LIN {X 0,Y 573.685,Z 492.708,A -85,B 0,C 180,E1 -2287.223,E2 -2287.223} C_VEL
LIN {X 0,Y 573.847,Z 485.027,A -85,B 0,C 180,E1 -2290.013,E2 -2290.013} C_VEL
LIN {X 0,Y 573.778,Z 480.732,A -85,B 0,C 180,E1 -2291.655,E2 -2291.655} C_VEL
LIN {X 0,Y 573.25,Z 477.707,A -85,B 0,C 180,E1 -2292.971,E2 -2292.971} C_VEL
LIN {X 0,Y 573.232,Z 477.709,A -85,B 0,C 180,E1 -2295.666,E2 -2295.666} C_VEL
LIN {X 0,Y 573.254,Z 477.706,A -85,B 0,C 180,E1 -2298.545,E2 -2298.545} C_VEL
LIN {X 0,Y 573.245,Z 477.706,A -85,B 0,C 180,E1 -2301.299,E2 -2301.299} C_VEL
LIN {X 0,Y 573.257,Z 477.705,A -85,B 0,C 180,E1 -2304.01,E2 -2304.01} C_VEL
LIN {X 0,Y 573.275,Z 477.704,A -85,B 0,C 180,E1 -2306.518,E2 -2306.518} C_VEL
LIN {X 0,Y 573.237,Z 477.707,A -85,B 0,C 180,E1 -2309.114,E2 -2309.114} C_VEL
LIN {X 0,Y 573.256,Z 477.706,A -85,B 0,C 180,E1 -2311.968,E2 -2311.968} C_VEL
LIN {X 0,Y 573.25,Z 477.705,A -85,B 0,C 180,E1 -2314.59,E2 -2314.59} C_VEL
LIN {X 0,Y 573.23,Z 477.709,A -85,B 0,C 180,E1 -2317.662,E2 -2317.662} C_VEL
LIN {X 0,Y 573.25,Z 477.706,A -85,B 0,C 180,E1 -2319.924,E2 -2319.924} C_VEL
LIN {X 0,Y 573.254,Z 477.707,A -85,B 0,C 180,E1 -2322.988,E2 -2322.988} C_VEL
LIN {X 0,Y 573.263,Z 477.704,A -85,B 0,C 180,E1 -2325.807,E2 -2325.807} C_VEL
LIN {X 0,Y 573.272,Z 477.703,A -85,B 0,C 180,E1 -2328.734,E2 -2328.734} C_VEL
LIN {X 0,Y 573.301,Z 477.7,A -85,B 0,C 180,E1 -2331.541,E2 -2331.541} C_VEL
LIN {X 0,Y 573.288,Z 477.7,A -85,B 0,C 180,E1 -2334.372,E2 -2334.372} C_VEL
LIN {X 0,Y 573.302,Z 477.699,A -85,B 0,C 180,E1 -2337.893,E2 -2337.893} C_VEL
LIN {X 0,Y 573.33,Z 477.697,A -85,B 0,C 180,E1 -2340.703,E2 -2340.703} C_VEL
LIN {X 0,Y 573.239,Z 477.707,A -85,B 0,C 180,E1 -2343.515,E2 -2343.515} C_VEL
LIN {X 0,Y 573.298,Z 477.699,A -85,B 0,C 180,E1 -2345.628,E2 -2345.628} C_VEL
LIN {X 0,Y 573.3,Z 477.7,A -85,B 0,C 180,E1 -2348.46,E2 -2348.46} C_VEL
LIN {X 0,Y 573.289,Z 477.701,A -85,B 0,C 180,E1 -2351.312,E2 -2351.312} C_VEL
LIN {X 0,Y 573.272,Z 477.702,A -85,B 0,C 180,E1 -2354.425,E2 -2354.425} C_VEL
LIN {X 0,Y 573.252,Z 477.707,A -85,B 0,C 180,E1 -2357.112,E2 -2357.112} C_VEL
LIN {X 0,Y 573.25,Z 477.706,A -85,B 0,C 180,E1 -2360.077,E2 -2360.077} C_VEL
LIN {X 0,Y 573.231,Z 477.708,A -85,B 0,C 180,E1 -2362.338,E2 -2362.338} C_VEL
LIN {X 0,Y 573.244,Z 477.706,A -85,B 0,C 180,E1 -2364.402,E2 -2364.402} C_VEL
LIN {X 0,Y 572.619,Z 477.786,A -85,B 0,C 180,E1 -2364.989,E2 -2364.989} C_VEL
LIN {X 0,Y 569.783,Z 478.14,A -85,B 0,C 180,E1 -2365.941,E2 -2365.941} C_VEL
LIN {X 0,Y 567.356,Z 478.442,A -85,B 0,C 180,E1 -2366.707,E2 -2366.707} C_VEL
LIN {X 0,Y 566.303,Z 478.572,A -85,B 0,C 180,E1 -2367.298,E2 -2367.298} C_VEL
LIN {X 0,Y 566.213,Z 478.581,A -85,B 0,C 180,E1 -2367.498,E2 -2367.498} C_VEL
LIN {X 0,Y 566.188,Z 478.585,A -85,B 0,C 180,E1 -2370.593,E2 -2370.593} C_VEL
LIN {X 0,Y 566.223,Z 478.58,A -85,B 0,C 180,E1 -2373.102,E2 -2373.102} C_VEL
LIN {X 0,Y 566.208,Z 478.584,A -85,B 0,C 180,E1 -2375.689,E2 -2375.689} C_VEL
LIN {X 0,Y 566.213,Z 478.581,A -85,B 0,C 180,E1 -2378.56,E2 -2378.56} C_VEL
LIN {X 0,Y 566.217,Z 478.582,A -85,B 0,C 180,E1 -2381.136,E2 -2381.136} C_VEL
LIN {X 0,Y 566.197,Z 478.584,A -85,B 0,C 180,E1 -2384.036,E2 -2384.036} C_VEL
LIN {X 0,Y 566.203,Z 478.584,A -85,B 0,C 180,E1 -2387.083,E2 -2387.083} C_VEL
LIN {X 0,Y 566.226,Z 478.581,A -85,B 0,C 180,E1 -2389.804,E2 -2389.804} C_VEL
LIN {X 0,Y 566.199,Z 478.584,A -85,B 0,C 180,E1 -2392.6,E2 -2392.6} C_VEL
LIN {X 0,Y 566.21,Z 478.582,A -85,B 0,C 180,E1 -2395.183,E2 -2395.183} C_VEL
LIN {X 0,Y 566.234,Z 478.581,A -85,B 0,C 180,E1 -2397.745,E2 -2397.745} C_VEL
LIN {X 0,Y 566.205,Z 478.582,A -85,B 0,C 180,E1 -2400.329,E2 -2400.329} C_VEL
LIN {X 0,Y 566.227,Z 478.579,A -85,B 0,C 180,E1 -2402.663,E2 -2402.663} C_VEL
LIN {X 0,Y 566.239,Z 478.578,A -85,B 0,C 180,E1 -2405.04,E2 -2405.04} C_VEL
LIN {X 0,Y 566.197,Z 478.583,A -85,B 0,C 180,E1 -2408.138,E2 -2408.138} C_VEL
LIN {X 0,Y 566.234,Z 478.578,A -85,B 0,C 180,E1 -2410.615,E2 -2410.615} C_VEL
LIN {X 0,Y 566.221,Z 478.582,A -85,B 0,C 180,E1 -2413.413,E2 -2413.413} C_VEL
LIN {X 0,Y 566.202,Z 478.584,A -85,B 0,C 180,E1 -2416.36,E2 -2416.36} C_VEL
LIN {X 0,Y 566.24,Z 478.58,A -85,B 0,C 180,E1 -2418.676,E2 -2418.676} C_VEL
LIN {X 0,Y 566.21,Z 478.582,A -85,B 0,C 180,E1 -2421.435,E2 -2421.435} C_VEL
LIN {X 0,Y 566.263,Z 478.577,A -85,B 0,C 180,E1 -2424.302,E2 -2424.302} C_VEL
LIN {X 0,Y 566.287,Z 478.573,A -85,B 0,C 180,E1 -2427.867,E2 -2427.867} C_VEL
LIN {X 0,Y 566.307,Z 478.571,A -85,B 0,C 180,E1 -2430.711,E2 -2430.711} C_VEL
LIN {X 0,Y 566.07,Z 478.602,A -85,B 0,C 180,E1 -2432.847,E2 -2432.847} C_VEL
LIN {X 0,Y 566.013,Z 478.622,A -85,B 0,C 180,E1 -2433.56,E2 -2433.56} C_VEL
LIN {X 0,Y 566.008,Z 480.702,A -85,B 0,C 180,E1 -2435.701,E2 -2435.701} C_VEL
LIN {X 0,Y 566.007,Z 483.486,A -85,B 0,C 180,E1 -2438.569,E2 -2438.569} C_VEL
LIN {X 0,Y 565.951,Z 486.311,A -85,B 0,C 180,E1 -2441.46,E2 -2441.46} C_VEL
LIN {X 0,Y 565.962,Z 489.393,A -85,B 0,C 180,E1 -2444.397,E2 -2444.397} C_VEL
LIN {X 0,Y 565.88,Z 492.716,A -85,B 0,C 180,E1 -2447.342,E2 -2447.342} C_VEL
LIN {X 0,Y 565.863,Z 496.182,A -85,B 0,C 180,E1 -2450.35,E2 -2450.35} C_VEL
LIN {X 0,Y 565.875,Z 498.386,A -85,B 0,C 180,E1 -2452.235,E2 -2452.235} C_VEL
LIN {X 0,Y 567.913,Z 507.747,A -85,B 0,C 180,E1 -2452.463,E2 -2452.463} C_VEL
LIN {X 0,Y 567.775,Z 523.279,A -85,B 0,C 180,E1 -2452.841,E2 -2452.841} C_VEL
LIN {X 0,Y 567.567,Z 537.926,A -85,B 0,C 180,E1 -2453.344,E2 -2453.344} C_VEL
LIN {X 0,Y 567.393,Z 551.473,A -85,B 0,C 180,E1 -2453.948,E2 -2453.948} C_VEL
LIN {X 0,Y 567.1,Z 565.407,A -85,B 0,C 180,E1 -2454.725,E2 -2454.725} C_VEL
LIN {X 0,Y 566.884,Z 578.74,A -85,B 0,C 180,E1 -2455.64,E2 -2455.64} C_VEL
LIN {X 0,Y 566.645,Z 591.048,A -85,B 0,C 180,E1 -2456.66,E2 -2456.66} C_VEL
LIN {X 0,Y 566.423,Z 601.892,A -85,B 0,C 180,E1 -2457.729,E2 -2457.729} C_VEL
LIN {X 0,Y 566.247,Z 612.279,A -85,B 0,C 180,E1 -2458.95,E2 -2458.95} C_VEL
LIN {X 0,Y 566.152,Z 621.068,A -85,B 0,C 180,E1 -2460.182,E2 -2460.182} C_VEL
LIN {X 0,Y 566.038,Z 629.621,A -85,B 0,C 180,E1 -2461.64,E2 -2461.64} C_VEL
LIN {X 0,Y 565.941,Z 636.591,A -85,B 0,C 180,E1 -2463.12,E2 -2463.12} C_VEL
LIN {X 0,Y 565.905,Z 641.383,A -85,B 0,C 180,E1 -2464.407,E2 -2464.407} C_VEL
LIN {X 0,Y 565.841,Z 645.15,A -85,B 0,C 180,E1 -2465.715,E2 -2465.715} C_VEL
LIN {X 0,Y 565.854,Z 647.11,A -85,B 0,C 180,E1 -2466.596,E2 -2466.596} C_VEL
LIN {X 0,Y 565.832,Z 648.638,A -85,B 0,C 180,E1 -2467.489,E2 -2467.489} C_VEL
LIN {X 0,Y 565.816,Z 649.833,A -85,B 0,C 180,E1 -2468.507,E2 -2468.507} C_VEL
LIN {X 0,Y 565.847,Z 650.418,A -85,B 0,C 180,E1 -2469.64,E2 -2469.64} C_VEL
LIN {X 0,Y 565.856,Z 650.112,A -85,B 0,C 180,E1 -2471.167,E2 -2471.167} C_VEL
LIN {X 0,Y 565.865,Z 649.261,A -85,B 0,C 180,E1 -2472.119,E2 -2472.119} C_VEL
LIN {X 0,Y 565.854,Z 647.882,A -85,B 0,C 180,E1 -2473.087,E2 -2473.087} C_VEL
LIN {X 0,Y 565.895,Z 644.84,A -85,B 0,C 180,E1 -2474.499,E2 -2474.499} C_VEL
LIN {X 0,Y 565.906,Z 640.511,A -85,B 0,C 180,E1 -2475.935,E2 -2475.935} C_VEL
LIN {X 0,Y 565.984,Z 636.025,A -85,B 0,C 180,E1 -2477.106,E2 -2477.106} C_VEL
LIN {X 0,Y 566.025,Z 629.345,A -85,B 0,C 180,E1 -2478.505,E2 -2478.505} C_VEL
LIN {X 0,Y 566.122,Z 621.792,A -85,B 0,C 180,E1 -2479.793,E2 -2479.793} C_VEL
LIN {X 0,Y 566.251,Z 612.523,A -85,B 0,C 180,E1 -2481.107,E2 -2481.107} C_VEL
LIN {X 0,Y 566.436,Z 602.143,A -85,B 0,C 180,E1 -2482.333,E2 -2482.333} C_VEL
LIN {X 0,Y 566.674,Z 590.668,A -85,B 0,C 180,E1 -2483.465,E2 -2483.465} C_VEL
LIN {X 0,Y 566.897,Z 578.806,A -85,B 0,C 180,E1 -2484.444,E2 -2484.444} C_VEL
LIN {X 0,Y 567.089,Z 567.299,A -85,B 0,C 180,E1 -2485.243,E2 -2485.243} C_VEL
LIN {X 0,Y 567.331,Z 553.585,A -85,B 0,C 180,E1 -2486.033,E2 -2486.033} C_VEL
LIN {X 0,Y 567.545,Z 539.884,A -85,B 0,C 180,E1 -2486.667,E2 -2486.667} C_VEL
LIN {X 0,Y 567.769,Z 524.257,A -85,B 0,C 180,E1 -2487.219,E2 -2487.219} C_VEL
LIN {X 0,Y 567.921,Z 508.637,A -85,B 0,C 180,E1 -2487.609,E2 -2487.609} C_VEL
LIN {X 0,Y 567.681,Z 506.099,A -85,B 0,C 180,E1 -2487.668,E2 -2487.668} C_VEL
LIN {X 0,Y 565.879,Z 498.374,A -85,B 0,C 180,E1 -2487.865,E2 -2487.865} C_VEL
LIN {X 0,Y 565.878,Z 495.432,A -85,B 0,C 180,E1 -2490.385,E2 -2490.385} C_VEL
LIN {X 0,Y 565.901,Z 491.926,A -85,B 0,C 180,E1 -2493.443,E2 -2493.443} C_VEL
LIN {X 0,Y 565.903,Z 489.271,A -85,B 0,C 180,E1 -2495.805,E2 -2495.805} C_VEL
LIN {X 0,Y 565.901,Z 486.833,A -85,B 0,C 180,E1 -2498.125,E2 -2498.125} C_VEL
LIN {X 0,Y 566.007,Z 484.648,A -85,B 0,C 180,E1 -2500.677,E2 -2500.677} C_VEL
LIN {X 0,Y 566.067,Z 482.103,A -85,B 0,C 180,E1 -2503.408,E2 -2503.408} C_VEL
LIN {X 0,Y 566.052,Z 479.234,A -85,B 0,C 180,E1 -2506.355,E2 -2506.355} C_VEL
LIN {X 0,Y 566.061,Z 478.604,A -85,B 0,C 180,E1 -2507.086,E2 -2507.086} C_VEL
LIN {X 0,Y 566.238,Z 478.574,A -85,B 0,C 180,E1 -2509.27,E2 -2509.27} C_VEL
LIN {X 0,Y 566.236,Z 478.58,A -85,B 0,C 180,E1 -2512.153,E2 -2512.153} C_VEL
LIN {X 0,Y 566.283,Z 478.567,A -85,B 0,C 180,E1 -2515.016,E2 -2515.016} C_VEL
LIN {X 0,Y 566.279,Z 478.574,A -85,B 0,C 180,E1 -2517.866,E2 -2517.866} C_VEL
LIN {X 0,Y 566.301,Z 478.565,A -85,B 0,C 180,E1 -2520.711,E2 -2520.711} C_VEL
LIN {X 0,Y 566.273,Z 478.57,A -85,B 0,C 180,E1 -2522.845,E2 -2522.845} C_VEL
LIN {X 0,Y 566.258,Z 478.573,A -85,B 0,C 180,E1 -2525.698,E2 -2525.698} C_VEL
LIN {X 0,Y 566.231,Z 478.575,A -85,B 0,C 180,E1 -2528.565,E2 -2528.565} C_VEL
LIN {X 0,Y 566.247,Z 478.574,A -85,B 0,C 180,E1 -2531.454,E2 -2531.454} C_VEL
LIN {X 0,Y 566.229,Z 478.578,A -85,B 0,C 180,E1 -2534.506,E2 -2534.506} C_VEL
LIN {X 0,Y 566.195,Z 478.579,A -85,B 0,C 180,E1 -2537.332,E2 -2537.332} C_VEL
LIN {X 0,Y 566.215,Z 478.581,A -85,B 0,C 180,E1 -2540.337,E2 -2540.337} C_VEL
LIN {X 0,Y 566.185,Z 478.579,A -85,B 0,C 180,E1 -2543.404,E2 -2543.404} C_VEL
LIN {X 0,Y 566.222,Z 478.577,A -85,B 0,C 180,E1 -2545.748,E2 -2545.748} C_VEL
LIN {X 0,Y 566.204,Z 478.585,A -85,B 0,C 180,E1 -2548.203,E2 -2548.203} C_VEL
LIN {X 0,Y 566.19,Z 478.58,A -85,B 0,C 180,E1 -2550.592,E2 -2550.592} C_VEL
LIN {X 0,Y 566.226,Z 478.575,A -85,B 0,C 180,E1 -2553.102,E2 -2553.102} C_VEL
LIN {X 0,Y 566.21,Z 478.585,A -85,B 0,C 180,E1 -2555.688,E2 -2555.688} C_VEL
LIN {X 0,Y 566.213,Z 478.575,A -85,B 0,C 180,E1 -2558.559,E2 -2558.559} C_VEL
LIN {X 0,Y 566.209,Z 478.581,A -85,B 0,C 180,E1 -2561.136,E2 -2561.136} C_VEL
LIN {X 0,Y 566.198,Z 478.581,A -85,B 0,C 180,E1 -2564.036,E2 -2564.036} C_VEL
LIN {X 0,Y 566.219,Z 478.637,A -85,B 0,C 180,E1 -2566.948,E2 -2566.948} C_VEL
LIN {X 0,Y 566.854,Z 483.368,A -85,B 0,C 180,E1 -2568.921,E2 -2568.921} C_VEL
LIN {X 0,Y 566.738,Z 489.853,A -85,B 0,C 180,E1 -2571.375,E2 -2571.375} C_VEL
LIN {X 0,Y 566.643,Z 498.211,A -85,B 0,C 180,E1 -2574.343,E2 -2574.343} C_VEL
LIN {X 0,Y 566.532,Z 505.812,A -85,B 0,C 180,E1 -2576.919,E2 -2576.919} C_VEL
LIN {X 0,Y 566.54,Z 513.738,A -85,B 0,C 180,E1 -2579.429,E2 -2579.429} C_VEL
LIN {X 0,Y 566.491,Z 521.49,A -85,B 0,C 180,E1 -2581.873,E2 -2581.873} C_VEL
LIN {X 0,Y 566.363,Z 530.126,A -85,B 0,C 180,E1 -2584.644,E2 -2584.644} C_VEL
LIN {X 0,Y 566.244,Z 538.819,A -85,B 0,C 180,E1 -2587.371,E2 -2587.371} C_VEL
LIN {X 0,Y 566.185,Z 547.483,A -85,B 0,C 180,E1 -2590.041,E2 -2590.041} C_VEL
LIN {X 0,Y 566.124,Z 554.42,A -85,B 0,C 180,E1 -2592.145,E2 -2592.145} C_VEL
LIN {X 0,Y 568.001,Z 563.349,A -85,B 0,C 180,E1 -2592.339,E2 -2592.339} C_VEL
LIN {X 0,Y 567.825,Z 577.885,A -85,B 0,C 180,E1 -2592.647,E2 -2592.647} C_VEL
LIN {X 0,Y 567.7,Z 592.206,A -85,B 0,C 180,E1 -2593.087,E2 -2593.087} C_VEL
LIN {X 0,Y 567.499,Z 605.82,A -85,B 0,C 180,E1 -2593.636,E2 -2593.636} C_VEL
LIN {X 0,Y 567.213,Z 620.1,A -85,B 0,C 180,E1 -2594.366,E2 -2594.366} C_VEL
LIN {X 0,Y 566.973,Z 633.394,A -85,B 0,C 180,E1 -2595.208,E2 -2595.208} C_VEL
LIN {X 0,Y 566.757,Z 646.161,A -85,B 0,C 180,E1 -2596.19,E2 -2596.19} C_VEL
LIN {X 0,Y 566.545,Z 657.97,A -85,B 0,C 180,E1 -2597.28,E2 -2597.28} C_VEL
LIN {X 0,Y 566.343,Z 667.9,A -85,B 0,C 180,E1 -2598.366,E2 -2598.366} C_VEL
LIN {X 0,Y 566.204,Z 677.618,A -85,B 0,C 180,E1 -2599.631,E2 -2599.631} C_VEL
LIN {X 0,Y 566.08,Z 685.72,A -85,B 0,C 180,E1 -2600.892,E2 -2600.892} C_VEL
LIN {X 0,Y 566.014,Z 692.424,A -85,B 0,C 180,E1 -2602.15,E2 -2602.15} C_VEL
LIN {X 0,Y 565.943,Z 698.606,A -85,B 0,C 180,E1 -2603.583,E2 -2603.583} C_VEL
LIN {X 0,Y 565.866,Z 703.384,A -85,B 0,C 180,E1 -2605.012,E2 -2605.012} C_VEL
LIN {X 0,Y 565.909,Z 706.888,A -85,B 0,C 180,E1 -2606.44,E2 -2606.44} C_VEL
LIN {X 0,Y 565.836,Z 709.192,A -85,B 0,C 180,E1 -2607.864,E2 -2607.864} C_VEL
LIN {X 0,Y 565.838,Z 710.349,A -85,B 0,C 180,E1 -2609.288,E2 -2609.288} C_VEL
LIN {X 0,Y 565.838,Z 710.349,A -85,B 0,C 180,E1 -2610.711,E2 -2610.711} C_VEL
LIN {X 0,Y 565.836,Z 709.191,A -85,B 0,C 180,E1 -2612.135,E2 -2612.135} C_VEL
LIN {X 0,Y 565.909,Z 706.888,A -85,B 0,C 180,E1 -2613.56,E2 -2613.56} C_VEL
LIN {X 0,Y 565.866,Z 703.386,A -85,B 0,C 180,E1 -2614.987,E2 -2614.987} C_VEL
LIN {X 0,Y 565.956,Z 699.926,A -85,B 0,C 180,E1 -2616.059,E2 -2616.059} C_VEL
LIN {X 0,Y 565.999,Z 694.09,A -85,B 0,C 180,E1 -2617.491,E2 -2617.491} C_VEL
LIN {X 0,Y 566.057,Z 686.733,A -85,B 0,C 180,E1 -2618.928,E2 -2618.928} C_VEL
LIN {X 0,Y 566.208,Z 678.861,A -85,B 0,C 180,E1 -2620.187,E2 -2620.187} C_VEL
LIN {X 0,Y 566.307,Z 669.395,A -85,B 0,C 180,E1 -2621.452,E2 -2621.452} C_VEL
LIN {X 0,Y 566.49,Z 659.754,A -85,B 0,C 180,E1 -2622.539,E2 -2622.539} C_VEL
LIN {X 0,Y 566.671,Z 648.299,A -85,B 0,C 180,E1 -2623.629,E2 -2623.629} C_VEL
LIN {X 0,Y 566.926,Z 635.681,A -85,B 0,C 180,E1 -2624.63,E2 -2624.63} C_VEL
LIN {X 0,Y 567.173,Z 623.252,A -85,B 0,C 180,E1 -2625.45,E2 -2625.45} C_VEL
LIN {X 0,Y 567.42,Z 609.779,A -85,B 0,C 180,E1 -2626.181,E2 -2626.181} C_VEL
LIN {X 0,Y 567.611,Z 596.065,A -85,B 0,C 180,E1 -2626.776,E2 -2626.776} C_VEL
LIN {X 0,Y 567.836,Z 580.741,A -85,B 0,C 180,E1 -2627.279,E2 -2627.279} C_VEL
LIN {X 0,Y 567.96,Z 565.547,A -85,B 0,C 180,E1 -2627.626,E2 -2627.626} C_VEL
LIN {X 0,Y 567.715,Z 561.412,A -85,B 0,C 180,E1 -2627.7,E2 -2627.7} C_VEL
LIN {X 0,Y 566.12,Z 554.385,A -85,B 0,C 180,E1 -2627.866,E2 -2627.866} C_VEL
LIN {X 0,Y 566.204,Z 545.01,A -85,B 0,C 180,E1 -2630.716,E2 -2630.716} C_VEL
LIN {X 0,Y 566.322,Z 535.108,A -85,B 0,C 180,E1 -2633.785,E2 -2633.785} C_VEL
LIN {X 0,Y 566.438,Z 525.894,A -85,B 0,C 180,E1 -2636.706,E2 -2636.706} C_VEL
LIN {X 0,Y 566.525,Z 517.758,A -85,B 0,C 180,E1 -2639.331,E2 -2639.331} C_VEL
LIN {X 0,Y 566.583,Z 508.792,A -85,B 0,C 180,E1 -2642.233,E2 -2642.233} C_VEL
LIN {X 0,Y 566.637,Z 500.309,A -85,B 0,C 180,E1 -2645.056,E2 -2645.056} C_VEL
LIN {X 0,Y 566.77,Z 492.32,A -85,B 0,C 180,E1 -2647.863,E2 -2647.863} C_VEL
LIN {X 0,Y 566.907,Z 486.184,A -85,B 0,C 180,E1 -2650.138,E2 -2650.138} C_VEL
LIN {X 0,Y 566.74,Z 481.588,A -85,B 0,C 180,E1 -2651.923,E2 -2651.923} C_VEL
LIN {X 0,Y 566.207,Z 478.585,A -85,B 0,C 180,E1 -2653.174,E2 -2653.174} C_VEL
LIN {X 0,Y 566.196,Z 478.584,A -85,B 0,C 180,E1 -2656.047,E2 -2656.047} C_VEL
LIN {X 0,Y 566.214,Z 478.584,A -85,B 0,C 180,E1 -2658.864,E2 -2658.864} C_VEL
LIN {X 0,Y 566.185,Z 478.585,A -85,B 0,C 180,E1 -2661.637,E2 -2661.637} C_VEL
LIN {X 0,Y 566.205,Z 478.585,A -85,B 0,C 180,E1 -2664.311,E2 -2664.311} C_VEL
LIN {X 0,Y 566.221,Z 478.581,A -85,B 0,C 180,E1 -2666.898,E2 -2666.898} C_VEL
LIN {X 0,Y 566.187,Z 478.585,A -85,B 0,C 180,E1 -2669.408,E2 -2669.408} C_VEL
LIN {X 0,Y 566.218,Z 478.583,A -85,B 0,C 180,E1 -2671.858,E2 -2671.858} C_VEL
LIN {X 0,Y 566.218,Z 478.582,A -85,B 0,C 180,E1 -2674.251,E2 -2674.251} C_VEL
LIN {X 0,Y 566.182,Z 478.586,A -85,B 0,C 180,E1 -2676.713,E2 -2676.713} C_VEL
LIN {X 0,Y 566.212,Z 478.584,A -85,B 0,C 180,E1 -2679.663,E2 -2679.663} C_VEL
LIN {X 0,Y 566.195,Z 478.584,A -85,B 0,C 180,E1 -2682.668,E2 -2682.668} C_VEL
LIN {X 0,Y 566.223,Z 478.581,A -85,B 0,C 180,E1 -2685.627,E2 -2685.627} C_VEL
LIN {X 0,Y 566.264,Z 478.576,A -85,B 0,C 180,E1 -2688.654,E2 -2688.654} C_VEL
LIN {X 0,Y 566.242,Z 478.579,A -85,B 0,C 180,E1 -2691.435,E2 -2691.435} C_VEL
LIN {X 0,Y 566.256,Z 478.576,A -85,B 0,C 180,E1 -2694.302,E2 -2694.302} C_VEL
LIN {X 0,Y 566.274,Z 478.574,A -85,B 0,C 180,E1 -2697.866,E2 -2697.866} C_VEL
LIN {X 0,Y 566.299,Z 478.573,A -85,B 0,C 180,E1 -2700.711,E2 -2700.711} C_VEL
LIN {X 0,Y 566.273,Z 478.576,A -85,B 0,C 180,E1 -2702.846,E2 -2702.846} C_VEL
LIN {X 0,Y 566.266,Z 478.576,A -85,B 0,C 180,E1 -2705.699,E2 -2705.699} C_VEL
LIN {X 0,Y 566.241,Z 478.578,A -85,B 0,C 180,E1 -2708.566,E2 -2708.566} C_VEL
LIN {X 0,Y 566.241,Z 478.58,A -85,B 0,C 180,E1 -2711.455,E2 -2711.455} C_VEL
LIN {X 0,Y 566.224,Z 478.58,A -85,B 0,C 180,E1 -2714.508,E2 -2714.508} C_VEL
LIN {X 0,Y 566.197,Z 478.585,A -85,B 0,C 180,E1 -2717.332,E2 -2717.332} C_VEL
LIN {X 0,Y 566.213,Z 478.584,A -85,B 0,C 180,E1 -2720.338,E2 -2720.338} C_VEL
LIN {X 0,Y 566.182,Z 478.586,A -85,B 0,C 180,E1 -2723.405,E2 -2723.405} C_VEL
LIN {X 0,Y 566.22,Z 478.582,A -85,B 0,C 180,E1 -2725.749,E2 -2725.749} C_VEL
LIN {X 0,Y 566.213,Z 478.581,A -85,B 0,C 180,E1 -2727.498,E2 -2727.498} C_VEL
LIN {X 0,Y 565.533,Z 478.669,A -85,B 0,C 180,E1 -2728.092,E2 -2728.092} C_VEL
LIN {X 0,Y 562.667,Z 479.024,A -85,B 0,C 180,E1 -2729.056,E2 -2729.056} C_VEL
LIN {X 0,Y 560.256,Z 479.324,A -85,B 0,C 180,E1 -2729.831,E2 -2729.831} C_VEL
LIN {X 0,Y 559.228,Z 479.453,A -85,B 0,C 180,E1 -2730.43,E2 -2730.43} C_VEL
LIN {X 0,Y 559.147,Z 479.461,A -85,B 0,C 180,E1 -2730.633,E2 -2730.633} C_VEL
LIN {X 0,Y 559.172,Z 479.461,A -85,B 0,C 180,E1 -2733.575,E2 -2733.575} C_VEL
LIN {X 0,Y 559.164,Z 479.459,A -85,B 0,C 180,E1 -2736.45,E2 -2736.45} C_VEL
LIN {X 0,Y 559.175,Z 479.458,A -85,B 0,C 180,E1 -2738.935,E2 -2738.935} C_VEL
LIN {X 0,Y 559.194,Z 479.456,A -85,B 0,C 180,E1 -2741.768,E2 -2741.768} C_VEL
LIN {X 0,Y 559.137,Z 479.465,A -85,B 0,C 180,E1 -2744.74,E2 -2744.74} C_VEL
LIN {X 0,Y 559.162,Z 479.46,A -85,B 0,C 180,E1 -2747.258,E2 -2747.258} C_VEL
LIN {X 0,Y 559.185,Z 479.459,A -85,B 0,C 180,E1 -2750.136,E2 -2750.136} C_VEL
LIN {X 0,Y 559.146,Z 479.461,A -85,B 0,C 180,E1 -2752.893,E2 -2752.893} C_VEL
LIN {X 0,Y 559.166,Z 479.459,A -85,B 0,C 180,E1 -2756.052,E2 -2756.052} C_VEL
LIN {X 0,Y 559.164,Z 479.462,A -85,B 0,C 180,E1 -2758.982,E2 -2758.982} C_VEL
LIN {X 0,Y 559.197,Z 479.457,A -85,B 0,C 180,E1 -2762.29,E2 -2762.29} C_VEL
LIN {X 0,Y 559.183,Z 479.457,A -85,B 0,C 180,E1 -2764.814,E2 -2764.814} C_VEL
LIN {X 0,Y 559.144,Z 479.464,A -85,B 0,C 180,E1 -2767.848,E2 -2767.848} C_VEL
LIN {X 0,Y 559.196,Z 479.455,A -85,B 0,C 180,E1 -2770.495,E2 -2770.495} C_VEL
LIN {X 0,Y 559.187,Z 479.458,A -85,B 0,C 180,E1 -2773.198,E2 -2773.198} C_VEL
LIN {X 0,Y 559.177,Z 479.458,A -85,B 0,C 180,E1 -2776.185,E2 -2776.185} C_VEL
LIN {X 0,Y 559.198,Z 479.456,A -85,B 0,C 180,E1 -2779.134,E2 -2779.134} C_VEL
LIN {X 0,Y 559.201,Z 479.457,A -85,B 0,C 180,E1 -2782.054,E2 -2782.054} C_VEL
LIN {X 0,Y 559.259,Z 479.447,A -85,B 0,C 180,E1 -2784.954,E2 -2784.954} C_VEL
LIN {X 0,Y 559.258,Z 479.449,A -85,B 0,C 180,E1 -2787.84,E2 -2787.84} C_VEL
LIN {X 0,Y 559.278,Z 479.447,A -85,B 0,C 180,E1 -2790.72,E2 -2790.72} C_VEL
LIN {X 0,Y 559.222,Z 479.455,A -85,B 0,C 180,E1 -2792.161,E2 -2792.161} C_VEL
LIN {X 0,Y 558.965,Z 479.489,A -85,B 0,C 180,E1 -2793.605,E2 -2793.605} C_VEL
LIN {X 0,Y 559.029,Z 480.704,A -85,B 0,C 180,E1 -2795.049,E2 -2795.049} C_VEL
LIN {X 0,Y 558.948,Z 483.516,A -85,B 0,C 180,E1 -2797.95,E2 -2797.95} C_VEL
LIN {X 0,Y 558.891,Z 486.716,A -85,B 0,C 180,E1 -2801.231,E2 -2801.231} C_VEL
LIN {X 0,Y 558.868,Z 489.964,A -85,B 0,C 180,E1 -2804.567,E2 -2804.567} C_VEL
LIN {X 0,Y 558.784,Z 493.315,A -85,B 0,C 180,E1 -2807.569,E2 -2807.569} C_VEL
LIN {X 0,Y 558.784,Z 495.908,A -85,B 0,C 180,E1 -2809.852,E2 -2809.852} C_VEL
LIN {X 0,Y 558.76,Z 498.383,A -85,B 0,C 180,E1 -2811.998,E2 -2811.998} C_VEL
LIN {X 0,Y 561.148,Z 508.688,A -85,B 0,C 180,E1 -2812.263,E2 -2812.263} C_VEL
LIN {X 0,Y 560.963,Z 524.384,A -85,B 0,C 180,E1 -2812.659,E2 -2812.659} C_VEL
LIN {X 0,Y 560.741,Z 538.446,A -85,B 0,C 180,E1 -2813.156,E2 -2813.156} C_VEL
LIN {X 0,Y 560.532,Z 552.742,A -85,B 0,C 180,E1 -2813.813,E2 -2813.813} C_VEL
LIN {X 0,Y 560.196,Z 565.775,A -85,B 0,C 180,E1 -2814.555,E2 -2814.555} C_VEL
LIN {X 0,Y 559.953,Z 578.637,A -85,B 0,C 180,E1 -2815.45,E2 -2815.45} C_VEL
LIN {X 0,Y 559.668,Z 590.88,A -85,B 0,C 180,E1 -2816.474,E2 -2816.474} C_VEL
LIN {X 0,Y 559.421,Z 602.026,A -85,B 0,C 180,E1 -2817.587,E2 -2817.587} C_VEL
LIN {X 0,Y 559.237,Z 611.688,A -85,B 0,C 180,E1 -2818.73,E2 -2818.73} C_VEL
LIN {X 0,Y 559.109,Z 620.61,A -85,B 0,C 180,E1 -2819.987,E2 -2819.987} C_VEL
LIN {X 0,Y 558.976,Z 628.063,A -85,B 0,C 180,E1 -2821.243,E2 -2821.243} C_VEL
LIN {X 0,Y 558.87,Z 635.316,A -85,B 0,C 180,E1 -2822.734,E2 -2822.734} C_VEL
LIN {X 0,Y 558.832,Z 639.886,A -85,B 0,C 180,E1 -2823.897,E2 -2823.897} C_VEL
LIN {X 0,Y 558.777,Z 644.382,A -85,B 0,C 180,E1 -2825.349,E2 -2825.349} C_VEL
LIN {X 0,Y 558.742,Z 646.785,A -85,B 0,C 180,E1 -2826.388,E2 -2826.388} C_VEL
LIN {X 0,Y 558.742,Z 648.836,A -85,B 0,C 180,E1 -2827.586,E2 -2827.586} C_VEL
LIN {X 0,Y 558.728,Z 650.152,A -85,B 0,C 180,E1 -2828.971,E2 -2828.971} C_VEL
LIN {X 0,Y 558.765,Z 650.475,A -85,B 0,C 180,E1 -2829.901,E2 -2829.901} C_VEL
LIN {X 0,Y 558.747,Z 650.229,A -85,B 0,C 180,E1 -2831.001,E2 -2831.001} C_VEL
LIN {X 0,Y 558.765,Z 649.322,A -85,B 0,C 180,E1 -2832.09,E2 -2832.09} C_VEL
LIN {X 0,Y 558.768,Z 647.836,A -85,B 0,C 180,E1 -2833.154,E2 -2833.154} C_VEL
LIN {X 0,Y 558.816,Z 644.306,A -85,B 0,C 180,E1 -2834.772,E2 -2834.772} C_VEL
LIN {X 0,Y 558.846,Z 639.734,A -85,B 0,C 180,E1 -2836.237,E2 -2836.237} C_VEL
LIN {X 0,Y 558.91,Z 634.283,A -85,B 0,C 180,E1 -2837.588,E2 -2837.588} C_VEL
LIN {X 0,Y 558.968,Z 627.376,A -85,B 0,C 180,E1 -2838.971,E2 -2838.971} C_VEL
LIN {X 0,Y 559.122,Z 618.859,A -85,B 0,C 180,E1 -2840.363,E2 -2840.363} C_VEL
LIN {X 0,Y 559.295,Z 609.787,A -85,B 0,C 180,E1 -2841.594,E2 -2841.594} C_VEL
LIN {X 0,Y 559.446,Z 599.524,A -85,B 0,C 180,E1 -2842.768,E2 -2842.768} C_VEL
LIN {X 0,Y 559.734,Z 588.444,A -85,B 0,C 180,E1 -2843.833,E2 -2843.833} C_VEL
LIN {X 0,Y 559.985,Z 575.856,A -85,B 0,C 180,E1 -2844.848,E2 -2844.848} C_VEL
LIN {X 0,Y 560.263,Z 562.904,A -85,B 0,C 180,E1 -2845.712,E2 -2845.712} C_VEL
LIN {X 0,Y 560.574,Z 548.926,A -85,B 0,C 180,E1 -2846.47,E2 -2846.47} C_VEL
LIN {X 0,Y 560.831,Z 535.224,A -85,B 0,C 180,E1 -2847.062,E2 -2847.062} C_VEL
LIN {X 0,Y 561.022,Z 520.305,A -85,B 0,C 180,E1 -2847.553,E2 -2847.553} C_VEL
LIN {X 0,Y 560.983,Z 507.559,A -85,B 0,C 180,E1 -2847.856,E2 -2847.856} C_VEL
LIN {X 0,Y 558.774,Z 498.375,A -85,B 0,C 180,E1 -2848.099,E2 -2848.099} C_VEL
LIN {X 0,Y 558.803,Z 495.464,A -85,B 0,C 180,E1 -2850.626,E2 -2850.626} C_VEL
LIN {X 0,Y 558.797,Z 491.786,A -85,B 0,C 180,E1 -2853.883,E2 -2853.883} C_VEL
LIN {X 0,Y 558.825,Z 488.836,A -85,B 0,C 180,E1 -2856.645,E2 -2856.645} C_VEL
LIN {X 0,Y 558.883,Z 486.46,A -85,B 0,C 180,E1 -2859.384,E2 -2859.384} C_VEL
LIN {X 0,Y 558.942,Z 484.504,A -85,B 0,C 180,E1 -2861.678,E2 -2861.678} C_VEL
LIN {X 0,Y 558.972,Z 482.223,A -85,B 0,C 180,E1 -2863.942,E2 -2863.942} C_VEL
LIN {X 0,Y 558.999,Z 480.105,A -85,B 0,C 180,E1 -2866.179,E2 -2866.179} C_VEL
LIN {X 0,Y 558.989,Z 479.484,A -85,B 0,C 180,E1 -2866.92,E2 -2866.92} C_VEL
LIN {X 0,Y 559.193,Z 479.451,A -85,B 0,C 180,E1 -2869.133,E2 -2869.133} C_VEL
LIN {X 0,Y 559.206,Z 479.457,A -85,B 0,C 180,E1 -2872.053,E2 -2872.053} C_VEL
LIN {X 0,Y 559.257,Z 479.443,A -85,B 0,C 180,E1 -2874.953,E2 -2874.953} C_VEL
LIN {X 0,Y 559.25,Z 479.45,A -85,B 0,C 180,E1 -2877.839,E2 -2877.839} C_VEL
LIN {X 0,Y 559.271,Z 479.441,A -85,B 0,C 180,E1 -2880.72,E2 -2880.72} C_VEL
LIN {X 0,Y 559.239,Z 479.446,A -85,B 0,C 180,E1 -2882.881,E2 -2882.881} C_VEL
LIN {X 0,Y 559.227,Z 479.449,A -85,B 0,C 180,E1 -2885.77,E2 -2885.77} C_VEL
LIN {X 0,Y 559.189,Z 479.454,A -85,B 0,C 180,E1 -2888.674,E2 -2888.674} C_VEL
LIN {X 0,Y 559.205,Z 479.45,A -85,B 0,C 180,E1 -2891.6,E2 -2891.6} C_VEL
LIN {X 0,Y 559.195,Z 479.455,A -85,B 0,C 180,E1 -2894.595,E2 -2894.595} C_VEL
LIN {X 0,Y 559.155,Z 479.455,A -85,B 0,C 180,E1 -2897.557,E2 -2897.557} C_VEL
LIN {X 0,Y 559.171,Z 479.453,A -85,B 0,C 180,E1 -2899.837,E2 -2899.837} C_VEL
LIN {X 0,Y 559.138,Z 479.462,A -85,B 0,C 180,E1 -2902.153,E2 -2902.153} C_VEL
LIN {X 0,Y 559.176,Z 479.452,A -85,B 0,C 180,E1 -2905.187,E2 -2905.187} C_VEL
LIN {X 0,Y 559.191,Z 479.454,A -85,B 0,C 180,E1 -2907.711,E2 -2907.711} C_VEL
LIN {X 0,Y 559.165,Z 479.461,A -85,B 0,C 180,E1 -2910.182,E2 -2910.182} C_VEL
LIN {X 0,Y 559.172,Z 479.453,A -85,B 0,C 180,E1 -2912.714,E2 -2912.714} C_VEL
LIN {X 0,Y 559.155,Z 479.459,A -85,B 0,C 180,E1 -2915.322,E2 -2915.322} C_VEL
LIN {X 0,Y 559.132,Z 479.461,A -85,B 0,C 180,E1 -2918.017,E2 -2918.017} C_VEL
LIN {X 0,Y 559.174,Z 479.454,A -85,B 0,C 180,E1 -2920.811,E2 -2920.811} C_VEL
LIN {X 0,Y 559.16,Z 479.46,A -85,B 0,C 180,E1 -2923.732,E2 -2923.732} C_VEL
LIN {X 0,Y 559.207,Z 479.62,A -85,B 0,C 180,E1 -2926.715,E2 -2926.715} C_VEL
LIN {X 0,Y 559.912,Z 484.669,A -85,B 0,C 180,E1 -2928.861,E2 -2928.861} C_VEL
LIN {X 0,Y 559.772,Z 490.529,A -85,B 0,C 180,E1 -2931.116,E2 -2931.116} C_VEL
LIN {X 0,Y 559.669,Z 498.038,A -85,B 0,C 180,E1 -2933.829,E2 -2933.829} C_VEL
LIN {X 0,Y 559.542,Z 505.515,A -85,B 0,C 180,E1 -2936.451,E2 -2936.451} C_VEL
LIN {X 0,Y 559.506,Z 514.744,A -85,B 0,C 180,E1 -2939.421,E2 -2939.421} C_VEL
LIN {X 0,Y 559.427,Z 523.922,A -85,B 0,C 180,E1 -2942.301,E2 -2942.301} C_VEL
LIN {X 0,Y 559.343,Z 531.602,A -85,B 0,C 180,E1 -2944.778,E2 -2944.778} C_VEL
LIN {X 0,Y 559.214,Z 540.056,A -85,B 0,C 180,E1 -2947.461,E2 -2947.461} C_VEL
LIN {X 0,Y 559.122,Z 549.866,A -85,B 0,C 180,E1 -2950.514,E2 -2950.514} C_VEL
LIN {X 0,Y 559.065,Z 554.423,A -85,B 0,C 180,E1 -2951.913,E2 -2951.913} C_VEL
LIN {X 0,Y 561.238,Z 564.229,A -85,B 0,C 180,E1 -2952.133,E2 -2952.133} C_VEL
LIN {X 0,Y 561.061,Z 579.832,A -85,B 0,C 180,E1 -2952.481,E2 -2952.481} C_VEL
LIN {X 0,Y 560.823,Z 595.201,A -85,B 0,C 180,E1 -2952.982,E2 -2952.982} C_VEL
LIN {X 0,Y 560.616,Z 609.769,A -85,B 0,C 180,E1 -2953.616,E2 -2953.616} C_VEL
LIN {X 0,Y 560.314,Z 623.243,A -85,B 0,C 180,E1 -2954.355,E2 -2954.355} C_VEL
LIN {X 0,Y 560.012,Z 636.463,A -85,B 0,C 180,E1 -2955.242,E2 -2955.242} C_VEL
LIN {X 0,Y 559.729,Z 648.289,A -85,B 0,C 180,E1 -2956.198,E2 -2956.198} C_VEL
LIN {X 0,Y 559.516,Z 659.748,A -85,B 0,C 180,E1 -2957.302,E2 -2957.302} C_VEL
LIN {X 0,Y 559.304,Z 669.389,A -85,B 0,C 180,E1 -2958.401,E2 -2958.401} C_VEL
LIN {X 0,Y 559.168,Z 678.856,A -85,B 0,C 180,E1 -2959.682,E2 -2959.682} C_VEL
LIN {X 0,Y 559.003,Z 686.732,A -85,B 0,C 180,E1 -2960.958,E2 -2960.958} C_VEL
LIN {X 0,Y 558.92,Z 694.088,A -85,B 0,C 180,E1 -2962.413,E2 -2962.413} C_VEL
LIN {X 0,Y 558.858,Z 699.922,A -85,B 0,C 180,E1 -2963.864,E2 -2963.864} C_VEL
LIN {X 0,Y 558.787,Z 703.385,A -85,B 0,C 180,E1 -2964.949,E2 -2964.949} C_VEL
LIN {X 0,Y 558.818,Z 706.889,A -85,B 0,C 180,E1 -2966.394,E2 -2966.394} C_VEL
LIN {X 0,Y 558.742,Z 709.192,A -85,B 0,C 180,E1 -2967.837,E2 -2967.837} C_VEL
LIN {X 0,Y 558.739,Z 710.349,A -85,B 0,C 180,E1 -2969.279,E2 -2969.279} C_VEL
LIN {X 0,Y 558.739,Z 710.349,A -85,B 0,C 180,E1 -2970.72,E2 -2970.72} C_VEL
LIN {X 0,Y 558.742,Z 709.191,A -85,B 0,C 180,E1 -2972.162,E2 -2972.162} C_VEL
LIN {X 0,Y 558.818,Z 706.888,A -85,B 0,C 180,E1 -2973.605,E2 -2973.605} C_VEL
LIN {X 0,Y 558.787,Z 703.387,A -85,B 0,C 180,E1 -2975.05,E2 -2975.05} C_VEL
LIN {X 0,Y 558.841,Z 698.61,A -85,B 0,C 180,E1 -2976.498,E2 -2976.498} C_VEL
LIN {X 0,Y 558.951,Z 692.425,A -85,B 0,C 180,E1 -2977.949,E2 -2977.949} C_VEL
LIN {X 0,Y 559.005,Z 684.651,A -85,B 0,C 180,E1 -2979.406,E2 -2979.406} C_VEL
LIN {X 0,Y 559.216,Z 676.373,A -85,B 0,C 180,E1 -2980.682,E2 -2980.682} C_VEL
LIN {X 0,Y 559.361,Z 666.397,A -85,B 0,C 180,E1 -2981.964,E2 -2981.964} C_VEL
LIN {X 0,Y 559.595,Z 656.194,A -85,B 0,C 180,E1 -2983.065,E2 -2983.065} C_VEL
LIN {X 0,Y 559.861,Z 644.027,A -85,B 0,C 180,E1 -2984.169,E2 -2984.169} C_VEL
LIN {X 0,Y 560.126,Z 631.702,A -85,B 0,C 180,E1 -2985.099,E2 -2985.099} C_VEL
LIN {X 0,Y 560.356,Z 618.526,A -85,B 0,C 180,E1 -2985.923,E2 -2985.923} C_VEL
LIN {X 0,Y 560.671,Z 603.846,A -85,B 0,C 180,E1 -2986.662,E2 -2986.662} C_VEL
LIN {X 0,Y 560.926,Z 588.994,A -85,B 0,C 180,E1 -2987.24,E2 -2987.24} C_VEL
LIN {X 0,Y 561.168,Z 573.463,A -85,B 0,C 180,E1 -2987.68,E2 -2987.68} C_VEL
LIN {X 0,Y 561.078,Z 563.107,A -85,B 0,C 180,E1 -2987.89,E2 -2987.89} C_VEL
LIN {X 0,Y 559.072,Z 554.409,A -85,B 0,C 180,E1 -2988.091,E2 -2988.091} C_VEL
LIN {X 0,Y 559.158,Z 545.01,A -85,B 0,C 180,E1 -2990.99,E2 -2990.99} C_VEL
LIN {X 0,Y 559.288,Z 535.108,A -85,B 0,C 180,E1 -2994.103,E2 -2994.103} C_VEL
LIN {X 0,Y 559.412,Z 526.443,A -85,B 0,C 180,E1 -2996.889,E2 -2996.889} C_VEL
LIN {X 0,Y 559.533,Z 517.018,A -85,B 0,C 180,E1 -2999.926,E2 -2999.926} C_VEL
LIN {X 0,Y 559.6,Z 508.573,A -85,B 0,C 180,E1 -3002.707,E2 -3002.707} C_VEL
LIN {X 0,Y 559.659,Z 500.932,A -85,B 0,C 180,E1 -3005.289,E2 -3005.289} C_VEL
LIN {X 0,Y 559.849,Z 492.223,A -85,B 0,C 180,E1 -3008.417,E2 -3008.417} C_VEL
LIN {X 0,Y 559.961,Z 486.087,A -85,B 0,C 180,E1 -3010.74,E2 -3010.74} C_VEL
LIN {X 0,Y 559.698,Z 482.447,A -85,B 0,C 180,E1 -3012.196,E2 -3012.196} C_VEL
LIN {X 0,Y 559.174,Z 479.459,A -85,B 0,C 180,E1 -3013.507,E2 -3013.507} C_VEL
LIN {X 0,Y 559.164,Z 479.461,A -85,B 0,C 180,E1 -3016.8,E2 -3016.8} C_VEL
LIN {X 0,Y 559.173,Z 479.459,A -85,B 0,C 180,E1 -3019.189,E2 -3019.189} C_VEL
LIN {X 0,Y 559.129,Z 479.467,A -85,B 0,C 180,E1 -3021.982,E2 -3021.982} C_VEL
LIN {X 0,Y 559.153,Z 479.461,A -85,B 0,C 180,E1 -3024.782,E2 -3024.782} C_VEL
LIN {X 0,Y 559.167,Z 479.461,A -85,B 0,C 180,E1 -3027.361,E2 -3027.361} C_VEL
LIN {X 0,Y 559.181,Z 479.457,A -85,B 0,C 180,E1 -3030.134,E2 -3030.134} C_VEL
LIN {X 0,Y 559.174,Z 479.461,A -85,B 0,C 180,E1 -3033.169,E2 -3033.169} C_VEL
LIN {X 0,Y 559.147,Z 479.463,A -85,B 0,C 180,E1 -3035.495,E2 -3035.495} C_VEL
LIN {X 0,Y 559.168,Z 479.461,A -85,B 0,C 180,E1 -3038.624,E2 -3038.624} C_VEL
LIN {X 0,Y 559.164,Z 479.461,A -85,B 0,C 180,E1 -3040.926,E2 -3040.926} C_VEL
LIN {X 0,Y 559.164,Z 479.462,A -85,B 0,C 180,E1 -3043.948,E2 -3043.948} C_VEL
LIN {X 0,Y 559.165,Z 479.462,A -85,B 0,C 180,E1 -3046.184,E2 -3046.184} C_VEL
LIN {X 0,Y 559.201,Z 479.455,A -85,B 0,C 180,E1 -3049.134,E2 -3049.134} C_VEL
LIN {X 0,Y 559.205,Z 479.455,A -85,B 0,C 180,E1 -3052.054,E2 -3052.054} C_VEL
LIN {X 0,Y 559.252,Z 479.449,A -85,B 0,C 180,E1 -3054.954,E2 -3054.954} C_VEL
LIN {X 0,Y 559.245,Z 479.45,A -85,B 0,C 180,E1 -3057.84,E2 -3057.84} C_VEL
LIN {X 0,Y 559.269,Z 479.448,A -85,B 0,C 180,E1 -3060.72,E2 -3060.72} C_VEL
LIN {X 0,Y 559.239,Z 479.453,A -85,B 0,C 180,E1 -3062.882,E2 -3062.882} C_VEL
LIN {X 0,Y 559.234,Z 479.452,A -85,B 0,C 180,E1 -3065.77,E2 -3065.77} C_VEL
LIN {X 0,Y 559.196,Z 479.456,A -85,B 0,C 180,E1 -3068.675,E2 -3068.675} C_VEL
LIN {X 0,Y 559.199,Z 479.458,A -85,B 0,C 180,E1 -3071.601,E2 -3071.601} C_VEL
LIN {X 0,Y 559.189,Z 479.457,A -85,B 0,C 180,E1 -3074.596,E2 -3074.596} C_VEL
LIN {X 0,Y 559.157,Z 479.461,A -85,B 0,C 180,E1 -3077.557,E2 -3077.557} C_VEL
LIN {X 0,Y 559.167,Z 479.459,A -85,B 0,C 180,E1 -3079.838,E2 -3079.838} C_VEL
LIN {X 0,Y 559.135,Z 479.463,A -85,B 0,C 180,E1 -3082.153,E2 -3082.153} C_VEL
LIN {X 0,Y 559.172,Z 479.459,A -85,B 0,C 180,E1 -3085.188,E2 -3085.188} C_VEL
LIN {X 0,Y 559.189,Z 479.457,A -85,B 0,C 180,E1 -3087.712,E2 -3087.712} C_VEL
LIN {X 0,Y 559.147,Z 479.461,A -85,B 0,C 180,E1 -3090.633,E2 -3090.633} C_VEL
LIN {X 0,Y 558.485,Z 479.546,A -85,B 0,C 180,E1 -3091.234,E2 -3091.234} C_VEL
LIN {X 0,Y 555.622,Z 479.902,A -85,B 0,C 180,E1 -3092.21,E2 -3092.21} C_VEL
LIN {X 0,Y 553.21,Z 480.201,A -85,B 0,C 180,E1 -3092.996,E2 -3092.996} C_VEL
LIN {X 0,Y 552.192,Z 480.331,A -85,B 0,C 180,E1 -3093.602,E2 -3093.602} C_VEL
LIN {X 0,Y 552.118,Z 480.336,A -85,B 0,C 180,E1 -3093.808,E2 -3093.808} C_VEL
LIN {X 0,Y 552.107,Z 480.339,A -85,B 0,C 180,E1 -3096.747,E2 -3096.747} C_VEL
LIN {X 0,Y 552.132,Z 480.336,A -85,B 0,C 180,E1 -3099.528,E2 -3099.528} C_VEL
LIN {X 0,Y 552.167,Z 480.333,A -85,B 0,C 180,E1 -3101.442,E2 -3101.442} C_VEL
LIN {X 0,Y 552.093,Z 480.342,A -85,B 0,C 180,E1 -3104.533,E2 -3104.533} C_VEL
LIN {X 0,Y 552.129,Z 480.337,A -85,B 0,C 180,E1 -3107.585,E2 -3107.585} C_VEL
LIN {X 0,Y 552.134,Z 480.335,A -85,B 0,C 180,E1 -3110.475,E2 -3110.475} C_VEL
LIN {X 0,Y 552.114,Z 480.339,A -85,B 0,C 180,E1 -3113.317,E2 -3113.317} C_VEL
LIN {X 0,Y 552.128,Z 480.336,A -85,B 0,C 180,E1 -3115.94,E2 -3115.94} C_VEL
LIN {X 0,Y 552.119,Z 480.337,A -85,B 0,C 180,E1 -3118.542,E2 -3118.542} C_VEL
LIN {X 0,Y 552.128,Z 480.337,A -85,B 0,C 180,E1 -3121.439,E2 -3121.439} C_VEL
LIN {X 0,Y 552.14,Z 480.336,A -85,B 0,C 180,E1 -3124.357,E2 -3124.357} C_VEL
LIN {X 0,Y 552.113,Z 480.34,A -85,B 0,C 180,E1 -3126.759,E2 -3126.759} C_VEL
LIN {X 0,Y 552.121,Z 480.338,A -85,B 0,C 180,E1 -3129.121,E2 -3129.121} C_VEL
LIN {X 0,Y 552.13,Z 480.336,A -85,B 0,C 180,E1 -3131.445,E2 -3131.445} C_VEL
LIN {X 0,Y 552.122,Z 480.337,A -85,B 0,C 180,E1 -3133.738,E2 -3133.738} C_VEL
LIN {X 0,Y 552.14,Z 480.335,A -85,B 0,C 180,E1 -3136.005,E2 -3136.005} C_VEL
LIN {X 0,Y 552.166,Z 480.332,A -85,B 0,C 180,E1 -3138.994,E2 -3138.994} C_VEL
LIN {X 0,Y 552.155,Z 480.335,A -85,B 0,C 180,E1 -3141.952,E2 -3141.952} C_VEL
LIN {X 0,Y 552.234,Z 480.322,A -85,B 0,C 180,E1 -3144.889,E2 -3144.889} C_VEL
LIN {X 0,Y 552.23,Z 480.324,A -85,B 0,C 180,E1 -3147.812,E2 -3147.812} C_VEL
LIN {X 0,Y 552.248,Z 480.322,A -85,B 0,C 180,E1 -3150.73,E2 -3150.73} C_VEL
LIN {X 0,Y 552.185,Z 480.331,A -85,B 0,C 180,E1 -3152.189,E2 -3152.189} C_VEL
LIN {X 0,Y 551.92,Z 480.366,A -85,B 0,C 180,E1 -3153.651,E2 -3153.651} C_VEL
LIN {X 0,Y 552.001,Z 480.709,A -85,B 0,C 180,E1 -3154.381,E2 -3154.381} C_VEL
LIN {X 0,Y 551.887,Z 483.526,A -85,B 0,C 180,E1 -3157.316,E2 -3157.316} C_VEL
LIN {X 0,Y 551.827,Z 486.353,A -85,B 0,C 180,E1 -3160.271,E2 -3160.271} C_VEL
LIN {X 0,Y 551.774,Z 488.513,A -85,B 0,C 180,E1 -3162.505,E2 -3162.505} C_VEL
LIN {X 0,Y 551.767,Z 490.641,A -85,B 0,C 180,E1 -3164.759,E2 -3164.759} C_VEL
LIN {X 0,Y 551.69,Z 493.914,A -85,B 0,C 180,E1 -3167.803,E2 -3167.803} C_VEL
LIN {X 0,Y 551.678,Z 496.517,A -85,B 0,C 180,E1 -3170.118,E2 -3170.118} C_VEL
LIN {X 0,Y 551.68,Z 498.378,A -85,B 0,C 180,E1 -3171.754,E2 -3171.754} C_VEL
LIN {X 0,Y 554.409,Z 510.538,A -85,B 0,C 180,E1 -3172.078,E2 -3172.078} C_VEL
LIN {X 0,Y 554.171,Z 525.848,A -85,B 0,C 180,E1 -3172.485,E2 -3172.485} C_VEL
LIN {X 0,Y 553.919,Z 540.141,A -85,B 0,C 180,E1 -3173.013,E2 -3173.013} C_VEL
LIN {X 0,Y 553.662,Z 553.69,A -85,B 0,C 180,E1 -3173.657,E2 -3173.657} C_VEL
LIN {X 0,Y 553.293,Z 567.657,A -85,B 0,C 180,E1 -3174.482,E2 -3174.482} C_VEL
LIN {X 0,Y 552.975,Z 580.794,A -85,B 0,C 180,E1 -3175.434,E2 -3175.434} C_VEL
LIN {X 0,Y 552.663,Z 593.231,A -85,B 0,C 180,E1 -3176.524,E2 -3176.524} C_VEL
LIN {X 0,Y 552.371,Z 604.166,A -85,B 0,C 180,E1 -3177.671,E2 -3177.671} C_VEL
LIN {X 0,Y 552.165,Z 614.192,A -85,B 0,C 180,E1 -3178.925,E2 -3178.925} C_VEL
LIN {X 0,Y 551.985,Z 623.311,A -85,B 0,C 180,E1 -3180.296,E2 -3180.296} C_VEL
LIN {X 0,Y 551.883,Z 630.929,A -85,B 0,C 180,E1 -3181.688,E2 -3181.688} C_VEL
LIN {X 0,Y 551.793,Z 637.62,A -85,B 0,C 180,E1 -3183.207,E2 -3183.207} C_VEL
LIN {X 0,Y 551.713,Z 642.232,A -85,B 0,C 180,E1 -3184.531,E2 -3184.531} C_VEL
LIN {X 0,Y 551.663,Z 645.808,A -85,B 0,C 180,E1 -3185.875,E2 -3185.875} C_VEL
LIN {X 0,Y 551.65,Z 647.648,A -85,B 0,C 180,E1 -3186.782,E2 -3186.782} C_VEL
LIN {X 0,Y 551.63,Z 649.154,A -85,B 0,C 180,E1 -3187.823,E2 -3187.823} C_VEL
LIN {X 0,Y 551.639,Z 650.179,A -85,B 0,C 180,E1 -3188.999,E2 -3188.999} C_VEL
LIN {X 0,Y 551.665,Z 650.404,A -85,B 0,C 180,E1 -3190.52,E2 -3190.52} C_VEL
LIN {X 0,Y 551.67,Z 649.923,A -85,B 0,C 180,E1 -3191.487,E2 -3191.487} C_VEL
LIN {X 0,Y 551.656,Z 648.93,A -85,B 0,C 180,E1 -3192.47,E2 -3192.47} C_VEL
LIN {X 0,Y 551.708,Z 646.352,A -85,B 0,C 180,E1 -3193.967,E2 -3193.967} C_VEL
LIN {X 0,Y 551.734,Z 642.328,A -85,B 0,C 180,E1 -3195.525,E2 -3195.525} C_VEL
LIN {X 0,Y 551.807,Z 636.965,A -85,B 0,C 180,E1 -3197.051,E2 -3197.051} C_VEL
LIN {X 0,Y 551.869,Z 630.3,A -85,B 0,C 180,E1 -3198.53,E2 -3198.53} C_VEL
LIN {X 0,Y 552.018,Z 622.214,A -85,B 0,C 180,E1 -3199.975,E2 -3199.975} C_VEL
LIN {X 0,Y 552.172,Z 614.099,A -85,B 0,C 180,E1 -3201.177,E2 -3201.177} C_VEL
LIN {X 0,Y 552.425,Z 603.645,A -85,B 0,C 180,E1 -3202.477,E2 -3202.477} C_VEL
LIN {X 0,Y 552.713,Z 592.448,A -85,B 0,C 180,E1 -3203.639,E2 -3203.639} C_VEL
LIN {X 0,Y 553.02,Z 580.496,A -85,B 0,C 180,E1 -3204.678,E2 -3204.678} C_VEL
LIN {X 0,Y 553.312,Z 567.755,A -85,B 0,C 180,E1 -3205.601,E2 -3205.601} C_VEL
LIN {X 0,Y 553.626,Z 554.247,A -85,B 0,C 180,E1 -3206.404,E2 -3206.404} C_VEL
LIN {X 0,Y 553.93,Z 539.612,A -85,B 0,C 180,E1 -3207.099,E2 -3207.099} C_VEL
LIN {X 0,Y 554.192,Z 524.199,A -85,B 0,C 180,E1 -3207.655,E2 -3207.655} C_VEL
LIN {X 0,Y 554.331,Z 509.306,A -85,B 0,C 180,E1 -3208.04,E2 -3208.04} C_VEL
LIN {X 0,Y 551.701,Z 498.373,A -85,B 0,C 180,E1 -3208.34,E2 -3208.34} C_VEL
LIN {X 0,Y 551.684,Z 495.303,A -85,B 0,C 180,E1 -3211.047,E2 -3211.047} C_VEL
LIN {X 0,Y 551.712,Z 492.543,A -85,B 0,C 180,E1 -3213.522,E2 -3213.522} C_VEL
LIN {X 0,Y 551.729,Z 490.146,A -85,B 0,C 180,E1 -3215.944,E2 -3215.944} C_VEL
LIN {X 0,Y 551.814,Z 488.011,A -85,B 0,C 180,E1 -3218.393,E2 -3218.393} C_VEL
LIN {X 0,Y 551.883,Z 486.121,A -85,B 0,C 180,E1 -3220.664,E2 -3220.664} C_VEL
LIN {X 0,Y 551.926,Z 483.832,A -85,B 0,C 180,E1 -3222.97,E2 -3222.97} C_VEL
LIN {X 0,Y 551.952,Z 481.022,A -85,B 0,C 180,E1 -3225.999,E2 -3225.999} C_VEL
LIN {X 0,Y 551.922,Z 480.365,A -85,B 0,C 180,E1 -3226.749,E2 -3226.749} C_VEL
LIN {X 0,Y 552.16,Z 480.328,A -85,B 0,C 180,E1 -3228.993,E2 -3228.993} C_VEL
LIN {X 0,Y 552.16,Z 480.335,A -85,B 0,C 180,E1 -3231.951,E2 -3231.951} C_VEL
LIN {X 0,Y 552.231,Z 480.318,A -85,B 0,C 180,E1 -3234.889,E2 -3234.889} C_VEL
LIN {X 0,Y 552.221,Z 480.326,A -85,B 0,C 180,E1 -3237.812,E2 -3237.812} C_VEL
LIN {X 0,Y 552.241,Z 480.317,A -85,B 0,C 180,E1 -3240.729,E2 -3240.729} C_VEL
LIN {X 0,Y 552.205,Z 480.323,A -85,B 0,C 180,E1 -3242.918,E2 -3242.918} C_VEL
LIN {X 0,Y 552.197,Z 480.324,A -85,B 0,C 180,E1 -3245.844,E2 -3245.844} C_VEL
LIN {X 0,Y 552.159,Z 480.331,A -85,B 0,C 180,E1 -3248.785,E2 -3248.785} C_VEL
LIN {X 0,Y 552.16,Z 480.327,A -85,B 0,C 180,E1 -3251.75,E2 -3251.75} C_VEL
LIN {X 0,Y 552.132,Z 480.338,A -85,B 0,C 180,E1 -3254.748,E2 -3254.748} C_VEL
LIN {X 0,Y 552.107,Z 480.333,A -85,B 0,C 180,E1 -3257.788,E2 -3257.788} C_VEL
LIN {X 0,Y 552.13,Z 480.333,A -85,B 0,C 180,E1 -3260.101,E2 -3260.101} C_VEL
LIN {X 0,Y 552.092,Z 480.343,A -85,B 0,C 180,E1 -3262.451,E2 -3262.451} C_VEL
LIN {X 0,Y 552.153,Z 480.327,A -85,B 0,C 180,E1 -3265.351,E2 -3265.351} C_VEL
LIN {X 0,Y 552.124,Z 480.339,A -85,B 0,C 180,E1 -3268.097,E2 -3268.097} C_VEL
LIN {X 0,Y 552.111,Z 480.335,A -85,B 0,C 180,E1 -3270.609,E2 -3270.609} C_VEL
LIN {X 0,Y 552.12,Z 480.333,A -85,B 0,C 180,E1 -3273.185,E2 -3273.185} C_VEL
LIN {X 0,Y 552.11,Z 480.34,A -85,B 0,C 180,E1 -3275.842,E2 -3275.842} C_VEL
LIN {X 0,Y 552.123,Z 480.333,A -85,B 0,C 180,E1 -3279.062,E2 -3279.062} C_VEL
LIN {X 0,Y 552.138,Z 480.336,A -85,B 0,C 180,E1 -3281.444,E2 -3281.444} C_VEL
LIN {X 0,Y 552.094,Z 480.339,A -85,B 0,C 180,E1 -3284.532,E2 -3284.532} C_VEL
LIN {X 0,Y 552.189,Z 480.457,A -85,B 0,C 180,E1 -3286.413,E2 -3286.413} C_VEL
LIN {X 0,Y 552.905,Z 485.516,A -85,B 0,C 180,E1 -3288.626,E2 -3288.626} C_VEL
LIN {X 0,Y 552.816,Z 491.194,A -85,B 0,C 180,E1 -3290.85,E2 -3290.85} C_VEL
LIN {X 0,Y 552.674,Z 499.094,A -85,B 0,C 180,E1 -3293.75,E2 -3293.75} C_VEL
LIN {X 0,Y 552.54,Z 506.605,A -85,B 0,C 180,E1 -3296.407,E2 -3296.407} C_VEL
LIN {X 0,Y 552.494,Z 515.75,A -85,B 0,C 180,E1 -3299.415,E2 -3299.415} C_VEL
LIN {X 0,Y 552.38,Z 524.846,A -85,B 0,C 180,E1 -3302.329,E2 -3302.329} C_VEL
LIN {X 0,Y 552.329,Z 532.146,A -85,B 0,C 180,E1 -3304.612,E2 -3304.612} C_VEL
LIN {X 0,Y 552.188,Z 541.294,A -85,B 0,C 180,E1 -3307.553,E2 -3307.553} C_VEL
LIN {X 0,Y 552.071,Z 551.197,A -85,B 0,C 180,E1 -3310.671,E2 -3310.671} C_VEL
LIN {X 0,Y 552.035,Z 554.391,A -85,B 0,C 180,E1 -3311.665,E2 -3311.665} C_VEL
LIN {X 0,Y 554.498,Z 565.349,A -85,B 0,C 180,E1 -3311.928,E2 -3311.928} C_VEL
LIN {X 0,Y 554.264,Z 580.703,A -85,B 0,C 180,E1 -3312.283,E2 -3312.283} C_VEL
LIN {X 0,Y 554.019,Z 595.546,A -85,B 0,C 180,E1 -3312.779,E2 -3312.779} C_VEL
LIN {X 0,Y 553.79,Z 609.771,A -85,B 0,C 180,E1 -3313.409,E2 -3313.409} C_VEL
LIN {X 0,Y 553.434,Z 623.245,A -85,B 0,C 180,E1 -3314.155,E2 -3314.155} C_VEL
LIN {X 0,Y 553.102,Z 636.464,A -85,B 0,C 180,E1 -3315.054,E2 -3315.054} C_VEL
LIN {X 0,Y 552.771,Z 649.349,A -85,B 0,C 180,E1 -3316.115,E2 -3316.115} C_VEL
LIN {X 0,Y 552.482,Z 661.507,A -85,B 0,C 180,E1 -3317.324,E2 -3317.324} C_VEL
LIN {X 0,Y 552.215,Z 671.483,A -85,B 0,C 180,E1 -3318.513,E2 -3318.513} C_VEL
LIN {X 0,Y 552.124,Z 680.086,A -85,B 0,C 180,E1 -3319.735,E2 -3319.735} C_VEL
LIN {X 0,Y 551.921,Z 687.742,A -85,B 0,C 180,E1 -3321.026,E2 -3321.026} C_VEL
LIN {X 0,Y 551.838,Z 694.089,A -85,B 0,C 180,E1 -3322.315,E2 -3322.315} C_VEL
LIN {X 0,Y 551.758,Z 699.607,A -85,B 0,C 180,E1 -3323.691,E2 -3323.691} C_VEL
LIN {X 0,Y 551.713,Z 703.385,A -85,B 0,C 180,E1 -3324.884,E2 -3324.884} C_VEL
LIN {X 0,Y 551.73,Z 706.889,A -85,B 0,C 180,E1 -3326.348,E2 -3326.348} C_VEL
LIN {X 0,Y 551.653,Z 709.191,A -85,B 0,C 180,E1 -3327.809,E2 -3327.809} C_VEL
LIN {X 0,Y 551.639,Z 710.349,A -85,B 0,C 180,E1 -3329.27,E2 -3329.27} C_VEL
LIN {X 0,Y 551.639,Z 710.348,A -85,B 0,C 180,E1 -3330.73,E2 -3330.73} C_VEL
LIN {X 0,Y 551.653,Z 709.19,A -85,B 0,C 180,E1 -3332.19,E2 -3332.19} C_VEL
LIN {X 0,Y 551.73,Z 706.888,A -85,B 0,C 180,E1 -3333.651,E2 -3333.651} C_VEL
LIN {X 0,Y 551.713,Z 703.387,A -85,B 0,C 180,E1 -3335.115,E2 -3335.115} C_VEL
LIN {X 0,Y 551.779,Z 698.611,A -85,B 0,C 180,E1 -3336.582,E2 -3336.582} C_VEL
LIN {X 0,Y 551.876,Z 692.425,A -85,B 0,C 180,E1 -3338.052,E2 -3338.052} C_VEL
LIN {X 0,Y 551.951,Z 684.65,A -85,B 0,C 180,E1 -3339.527,E2 -3339.527} C_VEL
LIN {X 0,Y 552.183,Z 676.373,A -85,B 0,C 180,E1 -3340.82,E2 -3340.82} C_VEL
LIN {X 0,Y 552.351,Z 666.397,A -85,B 0,C 180,E1 -3342.118,E2 -3342.118} C_VEL
LIN {X 0,Y 552.608,Z 656.194,A -85,B 0,C 180,E1 -3343.233,E2 -3343.233} C_VEL
LIN {X 0,Y 552.906,Z 644.027,A -85,B 0,C 180,E1 -3344.351,E2 -3344.351} C_VEL
LIN {X 0,Y 553.24,Z 631.456,A -85,B 0,C 180,E1 -3345.309,E2 -3345.309} C_VEL
LIN {X 0,Y 553.513,Z 618.524,A -85,B 0,C 180,E1 -3346.125,E2 -3346.125} C_VEL
LIN {X 0,Y 553.855,Z 603.844,A -85,B 0,C 180,E1 -3346.873,E2 -3346.873} C_VEL
LIN {X 0,Y 554.153,Z 588.572,A -85,B 0,C 180,E1 -3347.473,E2 -3347.473} C_VEL
LIN {X 0,Y 554.379,Z 572.683,A -85,B 0,C 180,E1 -3347.923,E2 -3347.923} C_VEL
LIN {X 0,Y 554.267,Z 564.008,A -85,B 0,C 180,E1 -3348.103,E2 -3348.103} C_VEL
LIN {X 0,Y 552.034,Z 554.391,A -85,B 0,C 180,E1 -3348.336,E2 -3348.336} C_VEL
LIN {X 0,Y 552.144,Z 545.01,A -85,B 0,C 180,E1 -3351.269,E2 -3351.269} C_VEL
LIN {X 0,Y 552.255,Z 536.346,A -85,B 0,C 180,E1 -3354.03,E2 -3354.03} C_VEL
LIN {X 0,Y 552.388,Z 528.853,A -85,B 0,C 180,E1 -3356.442,E2 -3356.442} C_VEL
LIN {X 0,Y 552.486,Z 519.922,A -85,B 0,C 180,E1 -3359.323,E2 -3359.323} C_VEL
LIN {X 0,Y 552.599,Z 511.042,A -85,B 0,C 180,E1 -3362.286,E2 -3362.286} C_VEL
LIN {X 0,Y 552.681,Z 503.355,A -85,B 0,C 180,E1 -3364.905,E2 -3364.905} C_VEL
LIN {X 0,Y 552.842,Z 494.787,A -85,B 0,C 180,E1 -3367.985,E2 -3367.985} C_VEL
LIN {X 0,Y 552.999,Z 488.437,A -85,B 0,C 180,E1 -3370.401,E2 -3370.401} C_VEL
LIN {X 0,Y 552.909,Z 484.765,A -85,B 0,C 180,E1 -3371.859,E2 -3371.859} C_VEL
LIN {X 0,Y 552.141,Z 480.334,A -85,B 0,C 180,E1 -3373.803,E2 -3373.803} C_VEL
LIN {X 0,Y 552.115,Z 480.34,A -85,B 0,C 180,E1 -3376.577,E2 -3376.577} C_VEL
LIN {X 0,Y 552.137,Z 480.336,A -85,B 0,C 180,E1 -3379.522,E2 -3379.522} C_VEL
LIN {X 0,Y 552.087,Z 480.342,A -85,B 0,C 180,E1 -3382.336,E2 -3382.336} C_VEL
LIN {X 0,Y 552.124,Z 480.337,A -85,B 0,C 180,E1 -3385.054,E2 -3385.054} C_VEL
LIN {X 0,Y 552.12,Z 480.338,A -85,B 0,C 180,E1 -3387.682,E2 -3387.682} C_VEL
LIN {X 0,Y 552.137,Z 480.334,A -85,B 0,C 180,E1 -3390.237,E2 -3390.237} C_VEL
LIN {X 0,Y 552.138,Z 480.336,A -85,B 0,C 180,E1 -3392.997,E2 -3392.997} C_VEL
LIN {X 0,Y 552.104,Z 480.341,A -85,B 0,C 180,E1 -3395.161,E2 -3395.161} C_VEL
LIN {X 0,Y 552.087,Z 480.343,A -85,B 0,C 180,E1 -3397.549,E2 -3397.549} C_VEL
LIN {X 0,Y 552.139,Z 480.335,A -85,B 0,C 180,E1 -3400.373,E2 -3400.373} C_VEL
LIN {X 0,Y 552.149,Z 480.335,A -85,B 0,C 180,E1 -3402.977,E2 -3402.977} C_VEL
LIN {X 0,Y 552.127,Z 480.337,A -85,B 0,C 180,E1 -3406.004,E2 -3406.004} C_VEL
LIN {X 0,Y 552.169,Z 480.331,A -85,B 0,C 180,E1 -3408.994,E2 -3408.994} C_VEL
LIN {X 0,Y 552.158,Z 480.333,A -85,B 0,C 180,E1 -3411.952,E2 -3411.952} C_VEL
LIN {X 0,Y 552.226,Z 480.324,A -85,B 0,C 180,E1 -3414.889,E2 -3414.889} C_VEL
LIN {X 0,Y 552.216,Z 480.325,A -85,B 0,C 180,E1 -3417.812,E2 -3417.812} C_VEL
LIN {X 0,Y 552.238,Z 480.324,A -85,B 0,C 180,E1 -3420.729,E2 -3420.729} C_VEL
LIN {X 0,Y 552.205,Z 480.328,A -85,B 0,C 180,E1 -3422.918,E2 -3422.918} C_VEL
LIN {X 0,Y 552.204,Z 480.328,A -85,B 0,C 180,E1 -3425.844,E2 -3425.844} C_VEL
LIN {X 0,Y 552.163,Z 480.331,A -85,B 0,C 180,E1 -3428.786,E2 -3428.786} C_VEL
LIN {X 0,Y 552.155,Z 480.334,A -85,B 0,C 180,E1 -3431.751,E2 -3431.751} C_VEL
LIN {X 0,Y 552.128,Z 480.337,A -85,B 0,C 180,E1 -3434.749,E2 -3434.749} C_VEL
LIN {X 0,Y 552.108,Z 480.339,A -85,B 0,C 180,E1 -3437.789,E2 -3437.789} C_VEL
LIN {X 0,Y 552.126,Z 480.337,A -85,B 0,C 180,E1 -3440.102,E2 -3440.102} C_VEL
LIN {X 0,Y 552.089,Z 480.342,A -85,B 0,C 180,E1 -3442.452,E2 -3442.452} C_VEL
LIN {X 0,Y 552.149,Z 480.334,A -85,B 0,C 180,E1 -3445.352,E2 -3445.352} C_VEL
LIN {X 0,Y 552.121,Z 480.339,A -85,B 0,C 180,E1 -3448.098,E2 -3448.098} C_VEL
LIN {X 0,Y 552.107,Z 480.339,A -85,B 0,C 180,E1 -3450.628,E2 -3450.628} C_VEL
LIN {X 0,Y 552.123,Z 480.337,A -85,B 0,C 180,E1 -3453.186,E2 -3453.186} C_VEL
LIN {X 0,Y 552.118,Z 480.336,A -85,B 0,C 180,E1 -3453.808,E2 -3453.808} C_VEL
LIN {X 0,Y 551.484,Z 480.417,A -85,B 0,C 180,E1 -3454.416,E2 -3454.416} C_VEL
LIN {X 0,Y 548.657,Z 480.772,A -85,B 0,C 180,E1 -3455.405,E2 -3455.405} C_VEL
LIN {X 0,Y 546.232,Z 481.074,A -85,B 0,C 180,E1 -3456.2,E2 -3456.2} C_VEL
LIN {X 0,Y 545.161,Z 481.206,A -85,B 0,C 180,E1 -3456.814,E2 -3456.814} C_VEL
LIN {X 0,Y 545.059,Z 481.218,A -85,B 0,C 180,E1 -3457.022,E2 -3457.022} C_VEL
LIN {X 0,Y 545.09,Z 481.215,A -85,B 0,C 180,E1 -3460.141,E2 -3460.141} C_VEL
LIN {X 0,Y 545.063,Z 481.217,A -85,B 0,C 180,E1 -3462.698,E2 -3462.698} C_VEL
LIN {X 0,Y 545.06,Z 481.216,A -85,B 0,C 180,E1 -3465.168,E2 -3465.168} C_VEL
LIN {X 0,Y 545.082,Z 481.216,A -85,B 0,C 180,E1 -3467.899,E2 -3467.899} C_VEL
LIN {X 0,Y 545.105,Z 481.21,A -85,B 0,C 180,E1 -3470.677,E2 -3470.677} C_VEL
LIN {X 0,Y 545.053,Z 481.219,A -85,B 0,C 180,E1 -3473.622,E2 -3473.622} C_VEL
LIN {X 0,Y 545.067,Z 481.216,A -85,B 0,C 180,E1 -3476.329,E2 -3476.329} C_VEL
LIN {X 0,Y 545.069,Z 481.217,A -85,B 0,C 180,E1 -3478.953,E2 -3478.953} C_VEL
LIN {X 0,Y 545.106,Z 481.211,A -85,B 0,C 180,E1 -3481.509,E2 -3481.509} C_VEL
LIN {X 0,Y 545.102,Z 481.212,A -85,B 0,C 180,E1 -3484.491,E2 -3484.491} C_VEL
LIN {X 0,Y 545.047,Z 481.218,A -85,B 0,C 180,E1 -3487.244,E2 -3487.244} C_VEL
LIN {X 0,Y 545.12,Z 481.208,A -85,B 0,C 180,E1 -3490.416,E2 -3490.416} C_VEL
LIN {X 0,Y 545.079,Z 481.215,A -85,B 0,C 180,E1 -3493.522,E2 -3493.522} C_VEL
LIN {X 0,Y 545.1,Z 481.212,A -85,B 0,C 180,E1 -3495.821,E2 -3495.821} C_VEL
LIN {X 0,Y 545.122,Z 481.21,A -85,B 0,C 180,E1 -3498.85,E2 -3498.85} C_VEL
LIN {X 0,Y 545.103,Z 481.213,A -85,B 0,C 180,E1 -3501.847,E2 -3501.847} C_VEL
LIN {X 0,Y 545.21,Z 481.197,A -85,B 0,C 180,E1 -3504.823,E2 -3504.823} C_VEL
LIN {X 0,Y 545.202,Z 481.2,A -85,B 0,C 180,E1 -3507.784,E2 -3507.784} C_VEL
LIN {X 0,Y 545.218,Z 481.198,A -85,B 0,C 180,E1 -3510.739,E2 -3510.739} C_VEL
LIN {X 0,Y 545.149,Z 481.208,A -85,B 0,C 180,E1 -3512.217,E2 -3512.217} C_VEL
LIN {X 0,Y 544.939,Z 481.435,A -85,B 0,C 180,E1 -3514.438,E2 -3514.438} C_VEL
LIN {X 0,Y 544.826,Z 484.275,A -85,B 0,C 180,E1 -3517.412,E2 -3517.412} C_VEL
LIN {X 0,Y 544.772,Z 487.126,A -85,B 0,C 180,E1 -3520.406,E2 -3520.406} C_VEL
LIN {X 0,Y 544.672,Z 490.007,A -85,B 0,C 180,E1 -3523.43,E2 -3523.43} C_VEL
LIN {X 0,Y 544.648,Z 492.143,A -85,B 0,C 180,E1 -3525.723,E2 -3525.723} C_VEL
LIN {X 0,Y 544.61,Z 494.513,A -85,B 0,C 180,E1 -3528.042,E2 -3528.042} C_VEL
LIN {X 0,Y 544.602,Z 497.124,A -85,B 0,C 180,E1 -3530.391,E2 -3530.391} C_VEL
LIN {X 0,Y 544.603,Z 498.381,A -85,B 0,C 180,E1 -3531.51,E2 -3531.51} C_VEL
LIN {X 0,Y 547.657,Z 511.678,A -85,B 0,C 180,E1 -3531.873,E2 -3531.873} C_VEL
LIN {X 0,Y 547.386,Z 526.526,A -85,B 0,C 180,E1 -3532.282,E2 -3532.282} C_VEL
LIN {X 0,Y 547.094,Z 540.68,A -85,B 0,C 180,E1 -3532.817,E2 -3532.817} C_VEL
LIN {X 0,Y 546.815,Z 554.313,A -85,B 0,C 180,E1 -3533.48,E2 -3533.48} C_VEL
LIN {X 0,Y 546.408,Z 568.012,A -85,B 0,C 180,E1 -3534.305,E2 -3534.305} C_VEL
LIN {X 0,Y 546.049,Z 581.409,A -85,B 0,C 180,E1 -3535.295,E2 -3535.295} C_VEL
LIN {X 0,Y 545.696,Z 593.554,A -85,B 0,C 180,E1 -3536.38,E2 -3536.38} C_VEL
LIN {X 0,Y 545.386,Z 604.283,A -85,B 0,C 180,E1 -3537.524,E2 -3537.524} C_VEL
LIN {X 0,Y 545.149,Z 614.035,A -85,B 0,C 180,E1 -3538.758,E2 -3538.758} C_VEL
LIN {X 0,Y 544.954,Z 623.471,A -85,B 0,C 180,E1 -3540.196,E2 -3540.196} C_VEL
LIN {X 0,Y 544.805,Z 631.198,A -85,B 0,C 180,E1 -3541.635,E2 -3541.635} C_VEL
LIN {X 0,Y 544.698,Z 637.167,A -85,B 0,C 180,E1 -3543,E2 -3543} C_VEL
LIN {X 0,Y 544.635,Z 641.836,A -85,B 0,C 180,E1 -3544.323,E2 -3544.323} C_VEL
LIN {X 0,Y 544.578,Z 645.293,A -85,B 0,C 180,E1 -3545.605,E2 -3545.605} C_VEL
LIN {X 0,Y 544.566,Z 647.832,A -85,B 0,C 180,E1 -3546.855,E2 -3546.855} C_VEL
LIN {X 0,Y 544.527,Z 649.675,A -85,B 0,C 180,E1 -3548.281,E2 -3548.281} C_VEL
LIN {X 0,Y 544.545,Z 650.335,A -85,B 0,C 180,E1 -3549.251,E2 -3549.251} C_VEL
LIN {X 0,Y 544.558,Z 650.43,A -85,B 0,C 180,E1 -3550.407,E2 -3550.407} C_VEL
LIN {X 0,Y 544.575,Z 649.902,A -85,B 0,C 180,E1 -3551.537,E2 -3551.537} C_VEL
LIN {X 0,Y 544.553,Z 647.953,A -85,B 0,C 180,E1 -3553.158,E2 -3553.158} C_VEL
LIN {X 0,Y 544.638,Z 644.564,A -85,B 0,C 180,E1 -3554.787,E2 -3554.787} C_VEL
LIN {X 0,Y 544.664,Z 640.168,A -85,B 0,C 180,E1 -3556.268,E2 -3556.268} C_VEL
LIN {X 0,Y 544.768,Z 635.059,A -85,B 0,C 180,E1 -3557.606,E2 -3557.606} C_VEL
LIN {X 0,Y 544.814,Z 628.235,A -85,B 0,C 180,E1 -3559.046,E2 -3559.046} C_VEL
LIN {X 0,Y 545.025,Z 619.619,A -85,B 0,C 180,E1 -3560.517,E2 -3560.517} C_VEL
LIN {X 0,Y 545.263,Z 610.267,A -85,B 0,C 180,E1 -3561.835,E2 -3561.835} C_VEL
LIN {X 0,Y 545.474,Z 600.302,A -85,B 0,C 180,E1 -3563.017,E2 -3563.017} C_VEL
LIN {X 0,Y 545.839,Z 589.01,A -85,B 0,C 180,E1 -3564.141,E2 -3564.141} C_VEL
LIN {X 0,Y 546.161,Z 576.745,A -85,B 0,C 180,E1 -3565.165,E2 -3565.165} C_VEL
LIN {X 0,Y 546.519,Z 563.223,A -85,B 0,C 180,E1 -3566.097,E2 -3566.097} C_VEL
LIN {X 0,Y 546.908,Z 550.128,A -85,B 0,C 180,E1 -3566.834,E2 -3566.834} C_VEL
LIN {X 0,Y 547.236,Z 536.035,A -85,B 0,C 180,E1 -3567.466,E2 -3567.466} C_VEL
LIN {X 0,Y 547.476,Z 520.745,A -85,B 0,C 180,E1 -3567.988,E2 -3567.988} C_VEL
LIN {X 0,Y 547.546,Z 510.428,A -85,B 0,C 180,E1 -3568.247,E2 -3568.247} C_VEL
LIN {X 0,Y 544.599,Z 498.388,A -85,B 0,C 180,E1 -3568.574,E2 -3568.574} C_VEL
LIN {X 0,Y 544.603,Z 495.142,A -85,B 0,C 180,E1 -3571.479,E2 -3571.479} C_VEL
LIN {X 0,Y 544.638,Z 492.586,A -85,B 0,C 180,E1 -3573.976,E2 -3573.976} C_VEL
LIN {X 0,Y 544.69,Z 490.407,A -85,B 0,C 180,E1 -3576.422,E2 -3576.422} C_VEL
LIN {X 0,Y 544.752,Z 488.36,A -85,B 0,C 180,E1 -3578.823,E2 -3578.823} C_VEL
LIN {X 0,Y 544.794,Z 486.251,A -85,B 0,C 180,E1 -3581.185,E2 -3581.185} C_VEL
LIN {X 0,Y 544.838,Z 484.024,A -85,B 0,C 180,E1 -3583.513,E2 -3583.513} C_VEL
LIN {X 0,Y 544.898,Z 481.944,A -85,B 0,C 180,E1 -3585.814,E2 -3585.814} C_VEL
LIN {X 0,Y 544.859,Z 481.251,A -85,B 0,C 180,E1 -3586.574,E2 -3586.574} C_VEL
LIN {X 0,Y 545.106,Z 481.208,A -85,B 0,C 180,E1 -3588.849,E2 -3588.849} C_VEL
LIN {X 0,Y 545.131,Z 481.209,A -85,B 0,C 180,E1 -3591.847,E2 -3591.847} C_VEL
LIN {X 0,Y 545.207,Z 481.193,A -85,B 0,C 180,E1 -3594.823,E2 -3594.823} C_VEL
LIN {X 0,Y 545.193,Z 481.202,A -85,B 0,C 180,E1 -3597.783,E2 -3597.783} C_VEL
LIN {X 0,Y 545.211,Z 481.193,A -85,B 0,C 180,E1 -3600.738,E2 -3600.738} C_VEL
LIN {X 0,Y 545.171,Z 481.2,A -85,B 0,C 180,E1 -3602.956,E2 -3602.956} C_VEL
LIN {X 0,Y 545.168,Z 481.199,A -85,B 0,C 180,E1 -3605.919,E2 -3605.919} C_VEL
LIN {X 0,Y 545.118,Z 481.209,A -85,B 0,C 180,E1 -3608.9,E2 -3608.9} C_VEL
LIN {X 0,Y 545.132,Z 481.202,A -85,B 0,C 180,E1 -3611.904,E2 -3611.904} C_VEL
LIN {X 0,Y 545.081,Z 481.214,A -85,B 0,C 180,E1 -3614.943,E2 -3614.943} C_VEL
LIN {X 0,Y 545.075,Z 481.21,A -85,B 0,C 180,E1 -3618.026,E2 -3618.026} C_VEL
LIN {X 0,Y 545.095,Z 481.213,A -85,B 0,C 180,E1 -3620.372,E2 -3620.372} C_VEL
LIN {X 0,Y 545.087,Z 481.208,A -85,B 0,C 180,E1 -3623.559,E2 -3623.559} C_VEL
LIN {X 0,Y 545.085,Z 481.213,A -85,B 0,C 180,E1 -3626,E2 -3626} C_VEL
LIN {X 0,Y 545.089,Z 481.209,A -85,B 0,C 180,E1 -3628.749,E2 -3628.749} C_VEL
LIN {X 0,Y 545.075,Z 481.215,A -85,B 0,C 180,E1 -3631.683,E2 -3631.683} C_VEL
LIN {X 0,Y 545.079,Z 481.21,A -85,B 0,C 180,E1 -3634.563,E2 -3634.563} C_VEL
LIN {X 0,Y 545.037,Z 481.219,A -85,B 0,C 180,E1 -3637.304,E2 -3637.304} C_VEL
LIN {X 0,Y 545.072,Z 481.211,A -85,B 0,C 180,E1 -3640.142,E2 -3640.142} C_VEL
LIN {X 0,Y 545.084,Z 481.216,A -85,B 0,C 180,E1 -3643.106,E2 -3643.106} C_VEL
LIN {X 0,Y 545.131,Z 481.339,A -85,B 0,C 180,E1 -3646.114,E2 -3646.114} C_VEL
LIN {X 0,Y 545.893,Z 486.244,A -85,B 0,C 180,E1 -3648.306,E2 -3648.306} C_VEL
LIN {X 0,Y 545.873,Z 491.854,A -85,B 0,C 180,E1 -3650.578,E2 -3650.578} C_VEL
LIN {X 0,Y 545.722,Z 498.21,A -85,B 0,C 180,E1 -3652.983,E2 -3652.983} C_VEL
LIN {X 0,Y 545.622,Z 505.299,A -85,B 0,C 180,E1 -3655.524,E2 -3655.524} C_VEL
LIN {X 0,Y 545.492,Z 514.325,A -85,B 0,C 180,E1 -3658.615,E2 -3658.615} C_VEL
LIN {X 0,Y 545.382,Z 523.2,A -85,B 0,C 180,E1 -3661.524,E2 -3661.524} C_VEL
LIN {X 0,Y 545.294,Z 532.475,A -85,B 0,C 180,E1 -3664.447,E2 -3664.447} C_VEL
LIN {X 0,Y 545.156,Z 541.294,A -85,B 0,C 180,E1 -3667.248,E2 -3667.248} C_VEL
LIN {X 0,Y 545.037,Z 550.752,A -85,B 0,C 180,E1 -3670.271,E2 -3670.271} C_VEL
LIN {X 0,Y 545.012,Z 554.415,A -85,B 0,C 180,E1 -3671.427,E2 -3671.427} C_VEL
LIN {X 0,Y 547.725,Z 566.255,A -85,B 0,C 180,E1 -3671.716,E2 -3671.716} C_VEL
LIN {X 0,Y 547.487,Z 581.827,A -85,B 0,C 180,E1 -3672.091,E2 -3672.091} C_VEL
LIN {X 0,Y 547.222,Z 595.87,A -85,B 0,C 180,E1 -3672.571,E2 -3672.571} C_VEL
LIN {X 0,Y 546.968,Z 609.773,A -85,B 0,C 180,E1 -3673.196,E2 -3673.196} C_VEL
LIN {X 0,Y 546.559,Z 623.247,A -85,B 0,C 180,E1 -3673.951,E2 -3673.951} C_VEL
LIN {X 0,Y 546.23,Z 635.526,A -85,B 0,C 180,E1 -3674.791,E2 -3674.791} C_VEL
LIN {X 0,Y 545.843,Z 648.291,A -85,B 0,C 180,E1 -3675.84,E2 -3675.84} C_VEL
LIN {X 0,Y 545.567,Z 659.748,A -85,B 0,C 180,E1 -3676.971,E2 -3676.971} C_VEL
LIN {X 0,Y 545.281,Z 669.388,A -85,B 0,C 180,E1 -3678.099,E2 -3678.099} C_VEL
LIN {X 0,Y 545.086,Z 678.855,A -85,B 0,C 180,E1 -3679.413,E2 -3679.413} C_VEL
LIN {X 0,Y 544.9,Z 686.734,A -85,B 0,C 180,E1 -3680.722,E2 -3680.722} C_VEL
LIN {X 0,Y 544.772,Z 694.089,A -85,B 0,C 180,E1 -3682.215,E2 -3682.215} C_VEL
LIN {X 0,Y 544.665,Z 699.95,A -85,B 0,C 180,E1 -3683.712,E2 -3683.712} C_VEL
LIN {X 0,Y 544.642,Z 703.385,A -85,B 0,C 180,E1 -3684.817,E2 -3684.817} C_VEL
LIN {X 0,Y 544.645,Z 706.888,A -85,B 0,C 180,E1 -3686.3,E2 -3686.3} C_VEL
LIN {X 0,Y 544.567,Z 709.191,A -85,B 0,C 180,E1 -3687.781,E2 -3687.781} C_VEL
LIN {X 0,Y 544.539,Z 710.348,A -85,B 0,C 180,E1 -3689.26,E2 -3689.26} C_VEL
LIN {X 0,Y 544.539,Z 710.348,A -85,B 0,C 180,E1 -3690.739,E2 -3690.739} C_VEL
LIN {X 0,Y 544.567,Z 709.189,A -85,B 0,C 180,E1 -3692.218,E2 -3692.218} C_VEL
LIN {X 0,Y 544.645,Z 706.887,A -85,B 0,C 180,E1 -3693.699,E2 -3693.699} C_VEL
LIN {X 0,Y 544.642,Z 703.387,A -85,B 0,C 180,E1 -3695.182,E2 -3695.182} C_VEL
LIN {X 0,Y 544.696,Z 698.611,A -85,B 0,C 180,E1 -3696.668,E2 -3696.668} C_VEL
LIN {X 0,Y 544.818,Z 692.424,A -85,B 0,C 180,E1 -3698.157,E2 -3698.157} C_VEL
LIN {X 0,Y 544.904,Z 684.649,A -85,B 0,C 180,E1 -3699.652,E2 -3699.652} C_VEL
LIN {X 0,Y 545.149,Z 676.372,A -85,B 0,C 180,E1 -3700.961,E2 -3700.961} C_VEL
LIN {X 0,Y 545.356,Z 666.396,A -85,B 0,C 180,E1 -3702.276,E2 -3702.276} C_VEL
LIN {X 0,Y 545.638,Z 656.193,A -85,B 0,C 180,E1 -3703.405,E2 -3703.405} C_VEL
LIN {X 0,Y 545.969,Z 644.027,A -85,B 0,C 180,E1 -3704.537,E2 -3704.537} C_VEL
LIN {X 0,Y 546.345,Z 631.656,A -85,B 0,C 180,E1 -3705.492,E2 -3705.492} C_VEL
LIN {X 0,Y 546.686,Z 618.522,A -85,B 0,C 180,E1 -3706.332,E2 -3706.332} C_VEL
LIN {X 0,Y 547.02,Z 603.842,A -85,B 0,C 180,E1 -3707.09,E2 -3707.09} C_VEL
LIN {X 0,Y 547.365,Z 589.221,A -85,B 0,C 180,E1 -3707.673,E2 -3707.673} C_VEL
LIN {X 0,Y 547.631,Z 574.051,A -85,B 0,C 180,E1 -3708.116,E2 -3708.116} C_VEL
LIN {X 0,Y 547.6,Z 565.477,A -85,B 0,C 180,E1 -3708.305,E2 -3708.305} C_VEL
LIN {X 0,Y 545.013,Z 554.373,A -85,B 0,C 180,E1 -3708.586,E2 -3708.586} C_VEL
LIN {X 0,Y 545.133,Z 543.772,A -85,B 0,C 180,E1 -3711.954,E2 -3711.954} C_VEL
LIN {X 0,Y 545.239,Z 535.061,A -85,B 0,C 180,E1 -3714.765,E2 -3714.765} C_VEL
LIN {X 0,Y 545.38,Z 525.935,A -85,B 0,C 180,E1 -3717.639,E2 -3717.639} C_VEL
LIN {X 0,Y 545.49,Z 517.031,A -85,B 0,C 180,E1 -3720.633,E2 -3720.633} C_VEL
LIN {X 0,Y 545.611,Z 509.711,A -85,B 0,C 180,E1 -3723.148,E2 -3723.148} C_VEL
LIN {X 0,Y 545.717,Z 502.187,A -85,B 0,C 180,E1 -3725.773,E2 -3725.773} C_VEL
LIN {X 0,Y 545.934,Z 494.454,A -85,B 0,C 180,E1 -3728.635,E2 -3728.635} C_VEL
LIN {X 0,Y 546.078,Z 488.31,A -85,B 0,C 180,E1 -3731.022,E2 -3731.022} C_VEL
LIN {X 0,Y 545.608,Z 484.144,A -85,B 0,C 180,E1 -3732.759,E2 -3732.759} C_VEL
LIN {X 0,Y 545.076,Z 481.215,A -85,B 0,C 180,E1 -3734.126,E2 -3734.126} C_VEL
LIN {X 0,Y 545.06,Z 481.218,A -85,B 0,C 180,E1 -3737.302,E2 -3737.302} C_VEL
LIN {X 0,Y 545.087,Z 481.216,A -85,B 0,C 180,E1 -3739.859,E2 -3739.859} C_VEL
LIN {X 0,Y 545.067,Z 481.218,A -85,B 0,C 180,E1 -3743.072,E2 -3743.072} C_VEL
LIN {X 0,Y 545.082,Z 481.215,A -85,B 0,C 180,E1 -3745.605,E2 -3745.605} C_VEL
LIN {X 0,Y 545.069,Z 481.216,A -85,B 0,C 180,E1 -3748.317,E2 -3748.317} C_VEL
LIN {X 0,Y 545.084,Z 481.214,A -85,B 0,C 180,E1 -3751.25,E2 -3751.25} C_VEL
LIN {X 0,Y 545.08,Z 481.216,A -85,B 0,C 180,E1 -3754,E2 -3754} C_VEL
LIN {X 0,Y 545.081,Z 481.215,A -85,B 0,C 180,E1 -3756.441,E2 -3756.441} C_VEL
LIN {X 0,Y 545.09,Z 481.216,A -85,B 0,C 180,E1 -3759.628,E2 -3759.628} C_VEL
LIN {X 0,Y 545.086,Z 481.213,A -85,B 0,C 180,E1 -3762.75,E2 -3762.75} C_VEL
LIN {X 0,Y 545.085,Z 481.214,A -85,B 0,C 180,E1 -3765.82,E2 -3765.82} C_VEL
LIN {X 0,Y 545.122,Z 481.209,A -85,B 0,C 180,E1 -3768.85,E2 -3768.85} C_VEL
LIN {X 0,Y 545.127,Z 481.21,A -85,B 0,C 180,E1 -3771.847,E2 -3771.847} C_VEL
LIN {X 0,Y 545.201,Z 481.198,A -85,B 0,C 180,E1 -3774.823,E2 -3774.823} C_VEL
LIN {X 0,Y 545.188,Z 481.201,A -85,B 0,C 180,E1 -3777.784,E2 -3777.784} C_VEL
LIN {X 0,Y 545.208,Z 481.2,A -85,B 0,C 180,E1 -3780.739,E2 -3780.739} C_VEL
LIN {X 0,Y 545.171,Z 481.204,A -85,B 0,C 180,E1 -3782.956,E2 -3782.956} C_VEL
LIN {X 0,Y 545.175,Z 481.204,A -85,B 0,C 180,E1 -3785.92,E2 -3785.92} C_VEL
LIN {X 0,Y 545.12,Z 481.209,A -85,B 0,C 180,E1 -3788.9,E2 -3788.9} C_VEL
LIN {X 0,Y 545.126,Z 481.208,A -85,B 0,C 180,E1 -3791.905,E2 -3791.905} C_VEL
LIN {X 0,Y 545.077,Z 481.216,A -85,B 0,C 180,E1 -3794.944,E2 -3794.944} C_VEL
LIN {X 0,Y 545.076,Z 481.216,A -85,B 0,C 180,E1 -3798.026,E2 -3798.026} C_VEL
LIN {X 0,Y 545.091,Z 481.214,A -85,B 0,C 180,E1 -3800.373,E2 -3800.373} C_VEL
LIN {X 0,Y 545.083,Z 481.215,A -85,B 0,C 180,E1 -3803.56,E2 -3803.56} C_VEL
LIN {X 0,Y 545.083,Z 481.215,A -85,B 0,C 180,E1 -3806.001,E2 -3806.001} C_VEL
LIN {X 0,Y 545.086,Z 481.212,A -85,B 0,C 180,E1 -3808.75,E2 -3808.75} C_VEL
LIN {X 0,Y 545.072,Z 481.216,A -85,B 0,C 180,E1 -3811.683,E2 -3811.683} C_VEL
LIN {X 0,Y 545.079,Z 481.215,A -85,B 0,C 180,E1 -3814.564,E2 -3814.564} C_VEL
LIN {X 0,Y 545.059,Z 481.218,A -85,B 0,C 180,E1 -3817.022,E2 -3817.022} C_VEL
LIN {X 0,Y 544.355,Z 481.306,A -85,B 0,C 180,E1 -3817.638,E2 -3817.638} C_VEL
LIN {X 0,Y 541.502,Z 481.658,A -85,B 0,C 180,E1 -3818.639,E2 -3818.639} C_VEL
LIN {X 0,Y 539.124,Z 481.957,A -85,B 0,C 180,E1 -3819.445,E2 -3819.445} C_VEL
LIN {X 0,Y 538.12,Z 482.083,A -85,B 0,C 180,E1 -3820.067,E2 -3820.067} C_VEL
LIN {X 0,Y 538.045,Z 482.088,A -85,B 0,C 180,E1 -3820.278,E2 -3820.278} C_VEL
LIN {X 0,Y 538.029,Z 482.092,A -85,B 0,C 180,E1 -3822.989,E2 -3822.989} C_VEL
LIN {X 0,Y 538.026,Z 482.093,A -85,B 0,C 180,E1 -3825.927,E2 -3825.927} C_VEL
LIN {X 0,Y 538.077,Z 482.088,A -85,B 0,C 180,E1 -3829.25,E2 -3829.25} C_VEL
LIN {X 0,Y 537.994,Z 482.098,A -85,B 0,C 180,E1 -3832.124,E2 -3832.124} C_VEL
LIN {X 0,Y 538.014,Z 482.094,A -85,B 0,C 180,E1 -3834.918,E2 -3834.918} C_VEL
LIN {X 0,Y 538.024,Z 482.094,A -85,B 0,C 180,E1 -3837.619,E2 -3837.619} C_VEL
LIN {X 0,Y 538.02,Z 482.093,A -85,B 0,C 180,E1 -3840.24,E2 -3840.24} C_VEL
LIN {X 0,Y 538.074,Z 482.086,A -85,B 0,C 180,E1 -3842.798,E2 -3842.798} C_VEL
LIN {X 0,Y 538.053,Z 482.09,A -85,B 0,C 180,E1 -3845.294,E2 -3845.294} C_VEL
LIN {X 0,Y 538.019,Z 482.094,A -85,B 0,C 180,E1 -3848.043,E2 -3848.043} C_VEL
LIN {X 0,Y 538.039,Z 482.091,A -85,B 0,C 180,E1 -3850.941,E2 -3850.941} C_VEL
LIN {X 0,Y 538.03,Z 482.094,A -85,B 0,C 180,E1 -3853.3,E2 -3853.3} C_VEL
LIN {X 0,Y 538.069,Z 482.089,A -85,B 0,C 180,E1 -3855.631,E2 -3855.631} C_VEL
LIN {X 0,Y 538.082,Z 482.086,A -85,B 0,C 180,E1 -3858.702,E2 -3858.702} C_VEL
LIN {X 0,Y 538.067,Z 482.088,A -85,B 0,C 180,E1 -3861.74,E2 -3861.74} C_VEL
LIN {X 0,Y 538.129,Z 482.081,A -85,B 0,C 180,E1 -3864.003,E2 -3864.003} C_VEL
LIN {X 0,Y 538.144,Z 482.078,A -85,B 0,C 180,E1 -3867.006,E2 -3867.006} C_VEL
LIN {X 0,Y 538.18,Z 482.074,A -85,B 0,C 180,E1 -3870,E2 -3870} C_VEL
LIN {X 0,Y 538.113,Z 482.084,A -85,B 0,C 180,E1 -3872.246,E2 -3872.246} C_VEL
LIN {X 0,Y 537.864,Z 482.162,A -85,B 0,C 180,E1 -3874.497,E2 -3874.497} C_VEL
LIN {X 0,Y 537.769,Z 485.023,A -85,B 0,C 180,E1 -3877.51,E2 -3877.51} C_VEL
LIN {X 0,Y 537.703,Z 487.877,A -85,B 0,C 180,E1 -3880.544,E2 -3880.544} C_VEL
LIN {X 0,Y 537.61,Z 490.781,A -85,B 0,C 180,E1 -3883.61,E2 -3883.61} C_VEL
LIN {X 0,Y 537.578,Z 492.956,A -85,B 0,C 180,E1 -3885.935,E2 -3885.935} C_VEL
LIN {X 0,Y 537.523,Z 495.188,A -85,B 0,C 180,E1 -3888.288,E2 -3888.288} C_VEL
LIN {X 0,Y 537.525,Z 498.371,A -85,B 0,C 180,E1 -3891.249,E2 -3891.249} C_VEL
LIN {X 0,Y 540.842,Z 511.848,A -85,B 0,C 180,E1 -3891.64,E2 -3891.64} C_VEL
LIN {X 0,Y 540.6,Z 527.264,A -85,B 0,C 180,E1 -3892.075,E2 -3892.075} C_VEL
LIN {X 0,Y 540.293,Z 541.509,A -85,B 0,C 180,E1 -3892.629,E2 -3892.629} C_VEL
LIN {X 0,Y 539.959,Z 554.755,A -85,B 0,C 180,E1 -3893.288,E2 -3893.288} C_VEL
LIN {X 0,Y 539.527,Z 568.401,A -85,B 0,C 180,E1 -3894.125,E2 -3894.125} C_VEL
LIN {X 0,Y 539.173,Z 580.939,A -85,B 0,C 180,E1 -3895.064,E2 -3895.064} C_VEL
LIN {X 0,Y 538.76,Z 591.979,A -85,B 0,C 180,E1 -3896.045,E2 -3896.045} C_VEL
LIN {X 0,Y 538.466,Z 602.767,A -85,B 0,C 180,E1 -3897.182,E2 -3897.182} C_VEL
LIN {X 0,Y 538.166,Z 613.023,A -85,B 0,C 180,E1 -3898.467,E2 -3898.467} C_VEL
LIN {X 0,Y 537.97,Z 621.688,A -85,B 0,C 180,E1 -3899.764,E2 -3899.764} C_VEL
LIN {X 0,Y 537.759,Z 629.049,A -85,B 0,C 180,E1 -3901.079,E2 -3901.079} C_VEL
LIN {X 0,Y 537.675,Z 635.152,A -85,B 0,C 180,E1 -3902.406,E2 -3902.406} C_VEL
LIN {X 0,Y 537.583,Z 640.214,A -85,B 0,C 180,E1 -3903.753,E2 -3903.753} C_VEL
LIN {X 0,Y 537.503,Z 644.282,A -85,B 0,C 180,E1 -3905.121,E2 -3905.121} C_VEL
LIN {X 0,Y 537.453,Z 646.402,A -85,B 0,C 180,E1 -3906.046,E2 -3906.046} C_VEL
LIN {X 0,Y 537.449,Z 648.248,A -85,B 0,C 180,E1 -3907.091,E2 -3907.091} C_VEL
LIN {X 0,Y 537.429,Z 649.733,A -85,B 0,C 180,E1 -3908.313,E2 -3908.313} C_VEL
LIN {X 0,Y 537.433,Z 650.465,A -85,B 0,C 180,E1 -3909.849,E2 -3909.849} C_VEL
LIN {X 0,Y 537.463,Z 650.341,A -85,B 0,C 180,E1 -3910.829,E2 -3910.829} C_VEL
LIN {X 0,Y 537.463,Z 649.683,A -85,B 0,C 180,E1 -3911.827,E2 -3911.827} C_VEL
LIN {X 0,Y 537.451,Z 648.369,A -85,B 0,C 180,E1 -3912.921,E2 -3912.921} C_VEL
LIN {X 0,Y 537.529,Z 645.549,A -85,B 0,C 180,E1 -3914.436,E2 -3914.436} C_VEL
LIN {X 0,Y 537.58,Z 641.405,A -85,B 0,C 180,E1 -3915.974,E2 -3915.974} C_VEL
LIN {X 0,Y 537.665,Z 636.215,A -85,B 0,C 180,E1 -3917.433,E2 -3917.433} C_VEL
LIN {X 0,Y 537.746,Z 629.374,A -85,B 0,C 180,E1 -3918.948,E2 -3918.948} C_VEL
LIN {X 0,Y 537.942,Z 621.099,A -85,B 0,C 180,E1 -3920.426,E2 -3920.426} C_VEL
LIN {X 0,Y 538.213,Z 611.236,A -85,B 0,C 180,E1 -3921.867,E2 -3921.867} C_VEL
LIN {X 0,Y 538.466,Z 601.104,A -85,B 0,C 180,E1 -3923.102,E2 -3923.102} C_VEL
LIN {X 0,Y 538.891,Z 589.363,A -85,B 0,C 180,E1 -3924.295,E2 -3924.295} C_VEL
LIN {X 0,Y 539.262,Z 576.621,A -85,B 0,C 180,E1 -3925.372,E2 -3925.372} C_VEL
LIN {X 0,Y 539.62,Z 564.465,A -85,B 0,C 180,E1 -3926.23,E2 -3926.23} C_VEL
LIN {X 0,Y 540.093,Z 550.093,A -85,B 0,C 180,E1 -3927.054,E2 -3927.054} C_VEL
LIN {X 0,Y 540.457,Z 535.044,A -85,B 0,C 180,E1 -3927.732,E2 -3927.732} C_VEL
LIN {X 0,Y 540.746,Z 519.623,A -85,B 0,C 180,E1 -3928.25,E2 -3928.25} C_VEL
LIN {X 0,Y 540.703,Z 511.249,A -85,B 0,C 180,E1 -3928.468,E2 -3928.468} C_VEL
LIN {X 0,Y 537.497,Z 498.365,A -85,B 0,C 180,E1 -3928.848,E2 -3928.848} C_VEL
LIN {X 0,Y 537.525,Z 495.123,A -85,B 0,C 180,E1 -3931.92,E2 -3931.92} C_VEL
LIN {X 0,Y 537.597,Z 492.825,A -85,B 0,C 180,E1 -3934.443,E2 -3934.443} C_VEL
LIN {X 0,Y 537.623,Z 490.677,A -85,B 0,C 180,E1 -3936.91,E2 -3936.91} C_VEL
LIN {X 0,Y 537.716,Z 488.652,A -85,B 0,C 180,E1 -3939.335,E2 -3939.335} C_VEL
LIN {X 0,Y 537.796,Z 485.667,A -85,B 0,C 180,E1 -3942.547,E2 -3942.547} C_VEL
LIN {X 0,Y 537.842,Z 482.879,A -85,B 0,C 180,E1 -3945.624,E2 -3945.624} C_VEL
LIN {X 0,Y 537.804,Z 482.198,A -85,B 0,C 180,E1 -3946.395,E2 -3946.395} C_VEL
LIN {X 0,Y 538.053,Z 482.088,A -85,B 0,C 180,E1 -3948.701,E2 -3948.701} C_VEL
LIN {X 0,Y 538.088,Z 482.085,A -85,B 0,C 180,E1 -3951.739,E2 -3951.739} C_VEL
LIN {X 0,Y 538.164,Z 482.071,A -85,B 0,C 180,E1 -3954.755,E2 -3954.755} C_VEL
LIN {X 0,Y 538.165,Z 482.077,A -85,B 0,C 180,E1 -3957.754,E2 -3957.754} C_VEL
LIN {X 0,Y 538.181,Z 482.069,A -85,B 0,C 180,E1 -3960.748,E2 -3960.748} C_VEL
LIN {X 0,Y 538.137,Z 482.076,A -85,B 0,C 180,E1 -3962.994,E2 -3962.994} C_VEL
LIN {X 0,Y 538.121,Z 482.076,A -85,B 0,C 180,E1 -3965.997,E2 -3965.997} C_VEL
LIN {X 0,Y 538.069,Z 482.089,A -85,B 0,C 180,E1 -3969.017,E2 -3969.017} C_VEL
LIN {X 0,Y 538.08,Z 482.08,A -85,B 0,C 180,E1 -3972.062,E2 -3972.062} C_VEL
LIN {X 0,Y 538.041,Z 482.089,A -85,B 0,C 180,E1 -3975.144,E2 -3975.144} C_VEL
LIN {X 0,Y 538.028,Z 482.09,A -85,B 0,C 180,E1 -3978.27,E2 -3978.27} C_VEL
LIN {X 0,Y 538.038,Z 482.092,A -85,B 0,C 180,E1 -3980.651,E2 -3980.651} C_VEL
LIN {X 0,Y 538.02,Z 482.09,A -85,B 0,C 180,E1 -3983.887,E2 -3983.887} C_VEL
LIN {X 0,Y 538.047,Z 482.091,A -85,B 0,C 180,E1 -3986.366,E2 -3986.366} C_VEL
LIN {X 0,Y 538.053,Z 482.085,A -85,B 0,C 180,E1 -3988.939,E2 -3988.939} C_VEL
LIN {X 0,Y 538.025,Z 482.095,A -85,B 0,C 180,E1 -3991.891,E2 -3991.891} C_VEL
LIN {X 0,Y 538.029,Z 482.088,A -85,B 0,C 180,E1 -3994.621,E2 -3994.621} C_VEL
LIN {X 0,Y 538.005,Z 482.094,A -85,B 0,C 180,E1 -3997.171,E2 -3997.171} C_VEL
LIN {X 0,Y 538.028,Z 482.092,A -85,B 0,C 180,E1 -3999.796,E2 -3999.796} C_VEL
LIN {X 0,Y 538.021,Z 482.093,A -85,B 0,C 180,E1 -4002.786,E2 -4002.786} C_VEL
LIN {X 0,Y 538.058,Z 482.217,A -85,B 0,C 180,E1 -4005.816,E2 -4005.816} C_VEL
LIN {X 0,Y 538.936,Z 487.693,A -85,B 0,C 180,E1 -4008.313,E2 -4008.313} C_VEL
LIN {X 0,Y 538.918,Z 492.535,A -85,B 0,C 180,E1 -4010.301,E2 -4010.301} C_VEL
LIN {X 0,Y 538.721,Z 499.891,A -85,B 0,C 180,E1 -4013.123,E2 -4013.123} C_VEL
LIN {X 0,Y 538.615,Z 505.762,A -85,B 0,C 180,E1 -4015.289,E2 -4015.289} C_VEL
LIN {X 0,Y 538.478,Z 515.071,A -85,B 0,C 180,E1 -4018.529,E2 -4018.529} C_VEL
LIN {X 0,Y 538.327,Z 524.126,A -85,B 0,C 180,E1 -4021.542,E2 -4021.542} C_VEL
LIN {X 0,Y 538.226,Z 532.667,A -85,B 0,C 180,E1 -4024.287,E2 -4024.287} C_VEL
LIN {X 0,Y 538.123,Z 542.531,A -85,B 0,C 180,E1 -4027.339,E2 -4027.339} C_VEL
LIN {X 0,Y 537.997,Z 551.197,A -85,B 0,C 180,E1 -4030.145,E2 -4030.145} C_VEL
LIN {X 0,Y 537.959,Z 554.419,A -85,B 0,C 180,E1 -4031.176,E2 -4031.176} C_VEL
LIN {X 0,Y 540.971,Z 567.648,A -85,B 0,C 180,E1 -4031.509,E2 -4031.509} C_VEL
LIN {X 0,Y 540.72,Z 582.694,A -85,B 0,C 180,E1 -4031.888,E2 -4031.888} C_VEL
LIN {X 0,Y 540.388,Z 597.991,A -85,B 0,C 180,E1 -4032.435,E2 -4032.435} C_VEL
LIN {X 0,Y 540.077,Z 611.597,A -85,B 0,C 180,E1 -4033.072,E2 -4033.072} C_VEL
LIN {X 0,Y 539.665,Z 624.772,A -85,B 0,C 180,E1 -4033.837,E2 -4033.837} C_VEL
LIN {X 0,Y 539.292,Z 637.445,A -85,B 0,C 180,E1 -4034.736,E2 -4034.736} C_VEL
LIN {X 0,Y 538.848,Z 650.377,A -85,B 0,C 180,E1 -4035.845,E2 -4035.845} C_VEL
LIN {X 0,Y 538.525,Z 661.507,A -85,B 0,C 180,E1 -4036.99,E2 -4036.99} C_VEL
LIN {X 0,Y 538.178,Z 671.728,A -85,B 0,C 180,E1 -4038.242,E2 -4038.242} C_VEL
LIN {X 0,Y 538.017,Z 681.294,A -85,B 0,C 180,E1 -4039.653,E2 -4039.653} C_VEL
LIN {X 0,Y 537.797,Z 688.749,A -85,B 0,C 180,E1 -4040.978,E2 -4040.978} C_VEL
LIN {X 0,Y 537.661,Z 695.7,A -85,B 0,C 180,E1 -4042.489,E2 -4042.489} C_VEL
LIN {X 0,Y 537.618,Z 701.161,A -85,B 0,C 180,E1 -4043.997,E2 -4043.997} C_VEL
LIN {X 0,Y 537.508,Z 705.291,A -85,B 0,C 180,E1 -4045.5,E2 -4045.5} C_VEL
LIN {X 0,Y 537.544,Z 708.185,A -85,B 0,C 180,E1 -4047.002,E2 -4047.002} C_VEL
LIN {X 0,Y 537.448,Z 709.91,A -85,B 0,C 180,E1 -4048.501,E2 -4048.501} C_VEL
LIN {X 0,Y 537.439,Z 710.5,A -85,B 0,C 180,E1 -4050,E2 -4050} C_VEL
LIN {X 0,Y 537.448,Z 709.909,A -85,B 0,C 180,E1 -4051.498,E2 -4051.498} C_VEL
LIN {X 0,Y 537.544,Z 708.183,A -85,B 0,C 180,E1 -4052.997,E2 -4052.997} C_VEL
LIN {X 0,Y 537.507,Z 705.291,A -85,B 0,C 180,E1 -4054.499,E2 -4054.499} C_VEL
LIN {X 0,Y 537.618,Z 701.166,A -85,B 0,C 180,E1 -4056.002,E2 -4056.002} C_VEL
LIN {X 0,Y 537.661,Z 695.703,A -85,B 0,C 180,E1 -4057.51,E2 -4057.51} C_VEL
LIN {X 0,Y 537.797,Z 688.749,A -85,B 0,C 180,E1 -4059.022,E2 -4059.022} C_VEL
LIN {X 0,Y 538.023,Z 680.088,A -85,B 0,C 180,E1 -4060.537,E2 -4060.537} C_VEL
LIN {X 0,Y 538.227,Z 670.538,A -85,B 0,C 180,E1 -4061.911,E2 -4061.911} C_VEL
LIN {X 0,Y 538.524,Z 661.513,A -85,B 0,C 180,E1 -4063.009,E2 -4063.009} C_VEL
LIN {X 0,Y 538.871,Z 649.364,A -85,B 0,C 180,E1 -4064.25,E2 -4064.25} C_VEL
LIN {X 0,Y 539.282,Z 637.508,A -85,B 0,C 180,E1 -4065.26,E2 -4065.26} C_VEL
LIN {X 0,Y 539.663,Z 624.781,A -85,B 0,C 180,E1 -4066.162,E2 -4066.162} C_VEL
LIN {X 0,Y 540.043,Z 611.605,A -85,B 0,C 180,E1 -4066.928,E2 -4066.928} C_VEL
LIN {X 0,Y 540.381,Z 598.011,A -85,B 0,C 180,E1 -4067.564,E2 -4067.564} C_VEL
LIN {X 0,Y 540.697,Z 583.37,A -85,B 0,C 180,E1 -4068.092,E2 -4068.092} C_VEL
LIN {X 0,Y 540.948,Z 568.031,A -85,B 0,C 180,E1 -4068.484,E2 -4068.484} C_VEL
LIN {X 0,Y 538.517,Z 556.866,A -85,B 0,C 180,E1 -4068.767,E2 -4068.767} C_VEL
LIN {X 0,Y 537.936,Z 554.354,A -85,B 0,C 180,E1 -4068.846,E2 -4068.846} C_VEL
LIN {X 0,Y 538.088,Z 544.629,A -85,B 0,C 180,E1 -4071.977,E2 -4071.977} C_VEL
LIN {X 0,Y 538.203,Z 536.061,A -85,B 0,C 180,E1 -4074.699,E2 -4074.699} C_VEL
LIN {X 0,Y 538.325,Z 527.562,A -85,B 0,C 180,E1 -4077.407,E2 -4077.407} C_VEL
LIN {X 0,Y 538.471,Z 518.371,A -85,B 0,C 180,E1 -4080.524,E2 -4080.524} C_VEL
LIN {X 0,Y 538.614,Z 510.185,A -85,B 0,C 180,E1 -4083.375,E2 -4083.375} C_VEL
LIN {X 0,Y 538.767,Z 501.726,A -85,B 0,C 180,E1 -4086.406,E2 -4086.406} C_VEL
LIN {X 0,Y 539.017,Z 494.311,A -85,B 0,C 180,E1 -4089.224,E2 -4089.224} C_VEL
LIN {X 0,Y 539.133,Z 490.118,A -85,B 0,C 180,E1 -4090.881,E2 -4090.881} C_VEL
LIN {X 0,Y 538.708,Z 485.757,A -85,B 0,C 180,E1 -4092.717,E2 -4092.717} C_VEL
LIN {X 0,Y 538.033,Z 482.094,A -85,B 0,C 180,E1 -4094.383,E2 -4094.383} C_VEL
LIN {X 0,Y 538.017,Z 482.095,A -85,B 0,C 180,E1 -4097.214,E2 -4097.214} C_VEL
LIN {X 0,Y 538.048,Z 482.091,A -85,B 0,C 180,E1 -4100.205,E2 -4100.205} C_VEL
LIN {X 0,Y 538.021,Z 482.095,A -85,B 0,C 180,E1 -4103.067,E2 -4103.067} C_VEL
LIN {X 0,Y 538.024,Z 482.093,A -85,B 0,C 180,E1 -4105.827,E2 -4105.827} C_VEL
LIN {X 0,Y 538.015,Z 482.095,A -85,B 0,C 180,E1 -4108.499,E2 -4108.499} C_VEL
LIN {X 0,Y 538.049,Z 482.091,A -85,B 0,C 180,E1 -4111.099,E2 -4111.099} C_VEL
LIN {X 0,Y 538.041,Z 482.091,A -85,B 0,C 180,E1 -4113.634,E2 -4113.634} C_VEL
LIN {X 0,Y 538.012,Z 482.096,A -85,B 0,C 180,E1 -4116.118,E2 -4116.118} C_VEL
LIN {X 0,Y 538.033,Z 482.092,A -85,B 0,C 180,E1 -4119.349,E2 -4119.349} C_VEL
LIN {X 0,Y 538.062,Z 482.087,A -85,B 0,C 180,E1 -4122.517,E2 -4122.517} C_VEL
LIN {X 0,Y 538.053,Z 482.09,A -85,B 0,C 180,E1 -4125.631,E2 -4125.631} C_VEL
LIN {X 0,Y 538.079,Z 482.087,A -85,B 0,C 180,E1 -4128.702,E2 -4128.702} C_VEL
LIN {X 0,Y 538.083,Z 482.088,A -85,B 0,C 180,E1 -4131.74,E2 -4131.74} C_VEL
LIN {X 0,Y 538.177,Z 482.073,A -85,B 0,C 180,E1 -4134.755,E2 -4134.755} C_VEL
LIN {X 0,Y 538.16,Z 482.076,A -85,B 0,C 180,E1 -4137.755,E2 -4137.755} C_VEL
LIN {X 0,Y 538.177,Z 482.075,A -85,B 0,C 180,E1 -4140.749,E2 -4140.749} C_VEL
LIN {X 0,Y 538.137,Z 482.08,A -85,B 0,C 180,E1 -4142.995,E2 -4142.995} C_VEL
LIN {X 0,Y 538.126,Z 482.082,A -85,B 0,C 180,E1 -4145.998,E2 -4145.998} C_VEL
LIN {X 0,Y 538.069,Z 482.087,A -85,B 0,C 180,E1 -4149.018,E2 -4149.018} C_VEL
LIN {X 0,Y 538.075,Z 482.086,A -85,B 0,C 180,E1 -4152.063,E2 -4152.063} C_VEL
LIN {X 0,Y 538.037,Z 482.093,A -85,B 0,C 180,E1 -4155.144,E2 -4155.144} C_VEL
LIN {X 0,Y 538.028,Z 482.093,A -85,B 0,C 180,E1 -4158.271,E2 -4158.271} C_VEL
LIN {X 0,Y 538.034,Z 482.092,A -85,B 0,C 180,E1 -4160.652,E2 -4160.652} C_VEL
LIN {X 0,Y 538.016,Z 482.095,A -85,B 0,C 180,E1 -4163.888,E2 -4163.888} C_VEL
LIN {X 0,Y 538.045,Z 482.089,A -85,B 0,C 180,E1 -4166.367,E2 -4166.367} C_VEL
LIN {X 0,Y 538.049,Z 482.089,A -85,B 0,C 180,E1 -4168.94,E2 -4168.94} C_VEL
LIN {X 0,Y 538.022,Z 482.093,A -85,B 0,C 180,E1 -4171.891,E2 -4171.891} C_VEL
LIN {X 0,Y 538.029,Z 482.093,A -85,B 0,C 180,E1 -4174.622,E2 -4174.622} C_VEL
LIN {X 0,Y 538.003,Z 482.097,A -85,B 0,C 180,E1 -4177.172,E2 -4177.172} C_VEL
LIN {X 0,Y 538.045,Z 482.088,A -85,B 0,C 180,E1 -4180.278,E2 -4180.278} C_VEL
LIN {X 0,Y 537.394,Z 482.171,A -85,B 0,C 180,E1 -4180.903,E2 -4180.903} C_VEL
LIN {X 0,Y 534.534,Z 482.531,A -85,B 0,C 180,E1 -4181.917,E2 -4181.917} C_VEL
LIN {X 0,Y 532.1,Z 482.836,A -85,B 0,C 180,E1 -4182.734,E2 -4182.734} C_VEL
LIN {X 0,Y 531.048,Z 482.965,A -85,B 0,C 180,E1 -4183.365,E2 -4183.365} C_VEL
LIN {X 0,Y 530.959,Z 482.974,A -85,B 0,C 180,E1 -4183.579,E2 -4183.579} C_VEL
LIN {X 0,Y 530.963,Z 482.972,A -85,B 0,C 180,E1 -4186.507,E2 -4186.507} C_VEL
LIN {X 0,Y 531.007,Z 482.967,A -85,B 0,C 180,E1 -4189.571,E2 -4189.571} C_VEL
LIN {X 0,Y 530.968,Z 482.972,A -85,B 0,C 180,E1 -4192.578,E2 -4192.578} C_VEL
LIN {X 0,Y 530.997,Z 482.969,A -85,B 0,C 180,E1 -4195.312,E2 -4195.312} C_VEL
LIN {X 0,Y 530.978,Z 482.971,A -85,B 0,C 180,E1 -4198.034,E2 -4198.034} C_VEL
LIN {X 0,Y 530.991,Z 482.968,A -85,B 0,C 180,E1 -4200.875,E2 -4200.875} C_VEL
LIN {X 0,Y 531.014,Z 482.967,A -85,B 0,C 180,E1 -4203.258,E2 -4203.258} C_VEL
LIN {X 0,Y 531,Z 482.968,A -85,B 0,C 180,E1 -4205.959,E2 -4205.959} C_VEL
LIN {X 0,Y 531.002,Z 482.969,A -85,B 0,C 180,E1 -4209.063,E2 -4209.063} C_VEL
LIN {X 0,Y 530.994,Z 482.969,A -85,B 0,C 180,E1 -4211.48,E2 -4211.48} C_VEL
LIN {X 0,Y 531.001,Z 482.968,A -85,B 0,C 180,E1 -4214.651,E2 -4214.651} C_VEL
LIN {X 0,Y 531.046,Z 482.964,A -85,B 0,C 180,E1 -4217.776,E2 -4217.776} C_VEL
LIN {X 0,Y 531.021,Z 482.966,A -85,B 0,C 180,E1 -4220.862,E2 -4220.862} C_VEL
LIN {X 0,Y 531.089,Z 482.958,A -85,B 0,C 180,E1 -4223.923,E2 -4223.923} C_VEL
LIN {X 0,Y 531.111,Z 482.954,A -85,B 0,C 180,E1 -4226.966,E2 -4226.966} C_VEL
LIN {X 0,Y 531.15,Z 482.95,A -85,B 0,C 180,E1 -4230,E2 -4230} C_VEL
LIN {X 0,Y 531.077,Z 482.96,A -85,B 0,C 180,E1 -4232.276,E2 -4232.276} C_VEL
LIN {X 0,Y 530.826,Z 482.993,A -85,B 0,C 180,E1 -4234.557,E2 -4234.557} C_VEL
LIN {X 0,Y 530.692,Z 485.784,A -85,B 0,C 180,E1 -4237.61,E2 -4237.61} C_VEL
LIN {X 0,Y 530.64,Z 488.67,A -85,B 0,C 180,E1 -4240.686,E2 -4240.686} C_VEL
LIN {X 0,Y 530.561,Z 491.595,A -85,B 0,C 180,E1 -4243.794,E2 -4243.794} C_VEL
LIN {X 0,Y 530.51,Z 493.823,A -85,B 0,C 180,E1 -4246.153,E2 -4246.153} C_VEL
LIN {X 0,Y 530.446,Z 496.032,A -85,B 0,C 180,E1 -4248.541,E2 -4248.541} C_VEL
LIN {X 0,Y 530.436,Z 498.379,A -85,B 0,C 180,E1 -4250.987,E2 -4250.987} C_VEL
LIN {X 0,Y 534.152,Z 513.488,A -85,B 0,C 180,E1 -4251.44,E2 -4251.44} C_VEL
LIN {X 0,Y 533.816,Z 528.62,A -85,B 0,C 180,E1 -4251.885,E2 -4251.885} C_VEL
LIN {X 0,Y 533.487,Z 542.865,A -85,B 0,C 180,E1 -4252.46,E2 -4252.46} C_VEL
LIN {X 0,Y 533.008,Z 557.314,A -85,B 0,C 180,E1 -4253.207,E2 -4253.207} C_VEL
LIN {X 0,Y 532.593,Z 570.288,A -85,B 0,C 180,E1 -4254.043,E2 -4254.043} C_VEL
LIN {X 0,Y 532.136,Z 583.839,A -85,B 0,C 180,E1 -4255.105,E2 -4255.105} C_VEL
LIN {X 0,Y 531.705,Z 595.548,A -85,B 0,C 180,E1 -4256.214,E2 -4256.214} C_VEL
LIN {X 0,Y 531.374,Z 605.735,A -85,B 0,C 180,E1 -4257.362,E2 -4257.362} C_VEL
LIN {X 0,Y 531.048,Z 616.356,A -85,B 0,C 180,E1 -4258.787,E2 -4258.787} C_VEL
LIN {X 0,Y 530.821,Z 625.062,A -85,B 0,C 180,E1 -4260.206,E2 -4260.206} C_VEL
LIN {X 0,Y 530.649,Z 632.877,A -85,B 0,C 180,E1 -4261.766,E2 -4261.766} C_VEL
LIN {X 0,Y 530.508,Z 639.421,A -85,B 0,C 180,E1 -4263.425,E2 -4263.425} C_VEL
LIN {X 0,Y 530.425,Z 643.504,A -85,B 0,C 180,E1 -4264.766,E2 -4264.766} C_VEL
LIN {X 0,Y 530.353,Z 646.539,A -85,B 0,C 180,E1 -4266.065,E2 -4266.065} C_VEL
LIN {X 0,Y 530.338,Z 648.969,A -85,B 0,C 180,E1 -4267.559,E2 -4267.559} C_VEL
LIN {X 0,Y 530.329,Z 649.933,A -85,B 0,C 180,E1 -4268.566,E2 -4268.566} C_VEL
LIN {X 0,Y 530.333,Z 650.449,A -85,B 0,C 180,E1 -4269.769,E2 -4269.769} C_VEL
LIN {X 0,Y 530.347,Z 649.952,A -85,B 0,C 180,E1 -4271.497,E2 -4271.497} C_VEL
LIN {X 0,Y 530.364,Z 648.987,A -85,B 0,C 180,E1 -4272.517,E2 -4272.517} C_VEL
LIN {X 0,Y 530.452,Z 645.958,A -85,B 0,C 180,E1 -4274.319,E2 -4274.319} C_VEL
LIN {X 0,Y 530.497,Z 641.361,A -85,B 0,C 180,E1 -4276.068,E2 -4276.068} C_VEL
LIN {X 0,Y 530.576,Z 636.331,A -85,B 0,C 180,E1 -4277.503,E2 -4277.503} C_VEL
LIN {X 0,Y 530.669,Z 629.626,A -85,B 0,C 180,E1 -4279.015,E2 -4279.015} C_VEL
LIN {X 0,Y 530.891,Z 621.207,A -85,B 0,C 180,E1 -4280.548,E2 -4280.548} C_VEL
LIN {X 0,Y 531.144,Z 612.962,A -85,B 0,C 180,E1 -4281.786,E2 -4281.786} C_VEL
LIN {X 0,Y 531.466,Z 602.376,A -85,B 0,C 180,E1 -4283.127,E2 -4283.127} C_VEL
LIN {X 0,Y 531.873,Z 590.934,A -85,B 0,C 180,E1 -4284.334,E2 -4284.334} C_VEL
LIN {X 0,Y 532.271,Z 578.774,A -85,B 0,C 180,E1 -4285.405,E2 -4285.405} C_VEL
LIN {X 0,Y 532.722,Z 565.822,A -85,B 0,C 180,E1 -4286.351,E2 -4286.351} C_VEL
LIN {X 0,Y 533.216,Z 551.962,A -85,B 0,C 180,E1 -4287.177,E2 -4287.177} C_VEL
LIN {X 0,Y 533.59,Z 538.356,A -85,B 0,C 180,E1 -4287.825,E2 -4287.825} C_VEL
LIN {X 0,Y 533.89,Z 523.25,A -85,B 0,C 180,E1 -4288.379,E2 -4288.379} C_VEL
LIN {X 0,Y 533.994,Z 512.681,A -85,B 0,C 180,E1 -4288.676,E2 -4288.676} C_VEL
LIN {X 0,Y 530.422,Z 498.392,A -85,B 0,C 180,E1 -4289.103,E2 -4289.103} C_VEL
LIN {X 0,Y 530.47,Z 495.342,A -85,B 0,C 180,E1 -4292.373,E2 -4292.373} C_VEL
LIN {X 0,Y 530.522,Z 493.075,A -85,B 0,C 180,E1 -4294.918,E2 -4294.918} C_VEL
LIN {X 0,Y 530.592,Z 490.46,A -85,B 0,C 180,E1 -4297.999,E2 -4297.999} C_VEL
LIN {X 0,Y 530.662,Z 488.095,A -85,B 0,C 180,E1 -4300.664,E2 -4300.664} C_VEL
LIN {X 0,Y 530.725,Z 485.969,A -85,B 0,C 180,E1 -4303.062,E2 -4303.062} C_VEL
LIN {X 0,Y 530.787,Z 483.858,A -85,B 0,C 180,E1 -4305.429,E2 -4305.429} C_VEL
LIN {X 0,Y 530.748,Z 483.143,A -85,B 0,C 180,E1 -4306.21,E2 -4306.21} C_VEL
LIN {X 0,Y 531.009,Z 482.967,A -85,B 0,C 180,E1 -4308.549,E2 -4308.549} C_VEL
LIN {X 0,Y 531.057,Z 482.959,A -85,B 0,C 180,E1 -4311.629,E2 -4311.629} C_VEL
LIN {X 0,Y 531.123,Z 482.948,A -85,B 0,C 180,E1 -4314.685,E2 -4314.685} C_VEL
LIN {X 0,Y 531.137,Z 482.953,A -85,B 0,C 180,E1 -4317.725,E2 -4317.725} C_VEL
LIN {X 0,Y 531.15,Z 482.944,A -85,B 0,C 180,E1 -4320.758,E2 -4320.758} C_VEL
LIN {X 0,Y 531.104,Z 482.953,A -85,B 0,C 180,E1 -4323.034,E2 -4323.034} C_VEL
LIN {X 0,Y 531.081,Z 482.953,A -85,B 0,C 180,E1 -4326.077,E2 -4326.077} C_VEL
LIN {X 0,Y 531.029,Z 482.966,A -85,B 0,C 180,E1 -4329.138,E2 -4329.138} C_VEL
LIN {X 0,Y 531.037,Z 482.958,A -85,B 0,C 180,E1 -4332.225,E2 -4332.225} C_VEL
LIN {X 0,Y 530.991,Z 482.965,A -85,B 0,C 180,E1 -4335.35,E2 -4335.35} C_VEL
LIN {X 0,Y 530.987,Z 482.971,A -85,B 0,C 180,E1 -4338.521,E2 -4338.521} C_VEL
LIN {X 0,Y 530.998,Z 482.965,A -85,B 0,C 180,E1 -4340.938,E2 -4340.938} C_VEL
LIN {X 0,Y 530.976,Z 482.973,A -85,B 0,C 180,E1 -4344.224,E2 -4344.224} C_VEL
LIN {X 0,Y 531.008,Z 482.964,A -85,B 0,C 180,E1 -4346.743,E2 -4346.743} C_VEL
LIN {X 0,Y 530.997,Z 482.964,A -85,B 0,C 180,E1 -4349.321,E2 -4349.321} C_VEL
LIN {X 0,Y 530.977,Z 482.972,A -85,B 0,C 180,E1 -4352.103,E2 -4352.103} C_VEL
LIN {X 0,Y 530.986,Z 482.965,A -85,B 0,C 180,E1 -4354.854,E2 -4354.854} C_VEL
LIN {X 0,Y 530.964,Z 482.974,A -85,B 0,C 180,E1 -4357.508,E2 -4357.508} C_VEL
LIN {X 0,Y 530.982,Z 482.965,A -85,B 0,C 180,E1 -4360.433,E2 -4360.433} C_VEL
LIN {X 0,Y 530.968,Z 482.974,A -85,B 0,C 180,E1 -4363.282,E2 -4363.282} C_VEL
LIN {X 0,Y 530.998,Z 482.998,A -85,B 0,C 180,E1 -4365.455,E2 -4365.455} C_VEL
LIN {X 0,Y 531.836,Z 487.821,A -85,B 0,C 180,E1 -4367.733,E2 -4367.733} C_VEL
LIN {X 0,Y 532.01,Z 492.319,A -85,B 0,C 180,E1 -4369.662,E2 -4369.662} C_VEL
LIN {X 0,Y 531.749,Z 499.601,A -85,B 0,C 180,E1 -4372.557,E2 -4372.557} C_VEL
LIN {X 0,Y 531.595,Z 507.103,A -85,B 0,C 180,E1 -4375.356,E2 -4375.356} C_VEL
LIN {X 0,Y 531.458,Z 516.019,A -85,B 0,C 180,E1 -4378.51,E2 -4378.51} C_VEL
LIN {X 0,Y 531.289,Z 525.053,A -85,B 0,C 180,E1 -4381.562,E2 -4381.562} C_VEL
LIN {X 0,Y 531.174,Z 534.172,A -85,B 0,C 180,E1 -4384.537,E2 -4384.537} C_VEL
LIN {X 0,Y 531.055,Z 543.443,A -85,B 0,C 180,E1 -4387.432,E2 -4387.432} C_VEL
LIN {X 0,Y 530.946,Z 552.662,A -85,B 0,C 180,E1 -4390.347,E2 -4390.347} C_VEL
LIN {X 0,Y 530.921,Z 554.428,A -85,B 0,C 180,E1 -4390.92,E2 -4390.92} C_VEL
LIN {X 0,Y 534.236,Z 568.855,A -85,B 0,C 180,E1 -4391.294,E2 -4391.294} C_VEL
LIN {X 0,Y 533.912,Z 584.316,A -85,B 0,C 180,E1 -4391.701,E2 -4391.701} C_VEL
LIN {X 0,Y 533.562,Z 599.912,A -85,B 0,C 180,E1 -4392.287,E2 -4392.287} C_VEL
LIN {X 0,Y 533.206,Z 613.361,A -85,B 0,C 180,E1 -4392.946,E2 -4392.946} C_VEL
LIN {X 0,Y 532.765,Z 626.194,A -85,B 0,C 180,E1 -4393.721,E2 -4393.721} C_VEL
LIN {X 0,Y 532.333,Z 639.349,A -85,B 0,C 180,E1 -4394.69,E2 -4394.69} C_VEL
LIN {X 0,Y 531.917,Z 650.375,A -85,B 0,C 180,E1 -4395.656,E2 -4395.656} C_VEL
LIN {X 0,Y 531.564,Z 661.507,A -85,B 0,C 180,E1 -4396.816,E2 -4396.816} C_VEL
LIN {X 0,Y 531.152,Z 672.268,A -85,B 0,C 180,E1 -4398.16,E2 -4398.16} C_VEL
LIN {X 0,Y 530.979,Z 681.294,A -85,B 0,C 180,E1 -4399.514,E2 -4399.514} C_VEL
LIN {X 0,Y 530.76,Z 688.749,A -85,B 0,C 180,E1 -4400.857,E2 -4400.857} C_VEL
LIN {X 0,Y 530.601,Z 695.7,A -85,B 0,C 180,E1 -4402.388,E2 -4402.388} C_VEL
LIN {X 0,Y 530.524,Z 701.161,A -85,B 0,C 180,E1 -4403.916,E2 -4403.916} C_VEL
LIN {X 0,Y 530.412,Z 705.291,A -85,B 0,C 180,E1 -4405.44,E2 -4405.44} C_VEL
LIN {X 0,Y 530.449,Z 708.185,A -85,B 0,C 180,E1 -4406.962,E2 -4406.962} C_VEL
LIN {X 0,Y 530.358,Z 709.91,A -85,B 0,C 180,E1 -4408.481,E2 -4408.481} C_VEL
LIN {X 0,Y 530.34,Z 710.5,A -85,B 0,C 180,E1 -4410,E2 -4410} C_VEL
LIN {X 0,Y 530.358,Z 709.908,A -85,B 0,C 180,E1 -4411.518,E2 -4411.518} C_VEL
LIN {X 0,Y 530.449,Z 708.182,A -85,B 0,C 180,E1 -4413.037,E2 -4413.037} C_VEL
LIN {X 0,Y 530.412,Z 705.29,A -85,B 0,C 180,E1 -4414.559,E2 -4414.559} C_VEL
LIN {X 0,Y 530.52,Z 701.167,A -85,B 0,C 180,E1 -4416.083,E2 -4416.083} C_VEL
LIN {X 0,Y 530.601,Z 695.703,A -85,B 0,C 180,E1 -4417.611,E2 -4417.611} C_VEL
LIN {X 0,Y 530.759,Z 688.748,A -85,B 0,C 180,E1 -4419.142,E2 -4419.142} C_VEL
LIN {X 0,Y 530.979,Z 681.296,A -85,B 0,C 180,E1 -4420.485,E2 -4420.485} C_VEL
LIN {X 0,Y 531.171,Z 671.96,A -85,B 0,C 180,E1 -4421.884,E2 -4421.884} C_VEL
LIN {X 0,Y 531.563,Z 661.513,A -85,B 0,C 180,E1 -4423.183,E2 -4423.183} C_VEL
LIN {X 0,Y 531.961,Z 649.365,A -85,B 0,C 180,E1 -4424.439,E2 -4424.439} C_VEL
LIN {X 0,Y 532.385,Z 637.131,A -85,B 0,C 180,E1 -4425.492,E2 -4425.492} C_VEL
LIN {X 0,Y 532.823,Z 623.262,A -85,B 0,C 180,E1 -4426.474,E2 -4426.474} C_VEL
LIN {X 0,Y 533.297,Z 609.786,A -85,B 0,C 180,E1 -4427.248,E2 -4427.248} C_VEL
LIN {X 0,Y 533.684,Z 596.387,A -85,B 0,C 180,E1 -4427.863,E2 -4427.863} C_VEL
LIN {X 0,Y 534.003,Z 580.742,A -85,B 0,C 180,E1 -4428.412,E2 -4428.412} C_VEL
LIN {X 0,Y 534.008,Z 567.461,A -85,B 0,C 180,E1 -4428.745,E2 -4428.745} C_VEL
LIN {X 0,Y 530.915,Z 554.375,A -85,B 0,C 180,E1 -4429.098,E2 -4429.098} C_VEL
LIN {X 0,Y 531.049,Z 544.953,A -85,B 0,C 180,E1 -4432.121,E2 -4432.121} C_VEL
LIN {X 0,Y 531.162,Z 535.76,A -85,B 0,C 180,E1 -4435.049,E2 -4435.049} C_VEL
LIN {X 0,Y 531.313,Z 526.69,A -85,B 0,C 180,E1 -4438.006,E2 -4438.006} C_VEL
LIN {X 0,Y 531.452,Z 518.798,A -85,B 0,C 180,E1 -4440.732,E2 -4440.732} C_VEL
LIN {X 0,Y 531.616,Z 510.665,A -85,B 0,C 180,E1 -4443.606,E2 -4443.606} C_VEL
LIN {X 0,Y 531.799,Z 502.803,A -85,B 0,C 180,E1 -4446.49,E2 -4446.49} C_VEL
LIN {X 0,Y 532.056,Z 495.389,A -85,B 0,C 180,E1 -4449.347,E2 -4449.347} C_VEL
LIN {X 0,Y 532.127,Z 490.494,A -85,B 0,C 180,E1 -4451.327,E2 -4451.327} C_VEL
LIN {X 0,Y 531.498,Z 485.625,A -85,B 0,C 180,E1 -4453.439,E2 -4453.439} C_VEL
LIN {X 0,Y 530.986,Z 482.97,A -85,B 0,C 180,E1 -4454.687,E2 -4454.687} C_VEL
LIN {X 0,Y 530.99,Z 482.971,A -85,B 0,C 180,E1 -4457.832,E2 -4457.832} C_VEL
LIN {X 0,Y 530.999,Z 482.969,A -85,B 0,C 180,E1 -4460.558,E2 -4460.558} C_VEL
LIN {X 0,Y 530.965,Z 482.972,A -85,B 0,C 180,E1 -4463.842,E2 -4463.842} C_VEL
LIN {X 0,Y 530.991,Z 482.97,A -85,B 0,C 180,E1 -4466.493,E2 -4466.493} C_VEL
LIN {X 0,Y 530.973,Z 482.972,A -85,B 0,C 180,E1 -4469.353,E2 -4469.353} C_VEL
LIN {X 0,Y 531.008,Z 482.965,A -85,B 0,C 180,E1 -4472.404,E2 -4472.404} C_VEL
LIN {X 0,Y 530.998,Z 482.968,A -85,B 0,C 180,E1 -4474.942,E2 -4474.942} C_VEL
LIN {X 0,Y 530.961,Z 482.973,A -85,B 0,C 180,E1 -4478.246,E2 -4478.246} C_VEL
LIN {X 0,Y 530.988,Z 482.97,A -85,B 0,C 180,E1 -4480.677,E2 -4480.677} C_VEL
LIN {X 0,Y 530.984,Z 482.972,A -85,B 0,C 180,E1 -4483.071,E2 -4483.071} C_VEL
LIN {X 0,Y 531.008,Z 482.968,A -85,B 0,C 180,E1 -4485.436,E2 -4485.436} C_VEL
LIN {X 0,Y 531.036,Z 482.964,A -85,B 0,C 180,E1 -4488.55,E2 -4488.55} C_VEL
LIN {X 0,Y 531.052,Z 482.963,A -85,B 0,C 180,E1 -4491.63,E2 -4491.63} C_VEL
LIN {X 0,Y 531.133,Z 482.95,A -85,B 0,C 180,E1 -4494.686,E2 -4494.686} C_VEL
LIN {X 0,Y 531.132,Z 482.952,A -85,B 0,C 180,E1 -4497.725,E2 -4497.725} C_VEL
LIN {X 0,Y 531.147,Z 482.951,A -85,B 0,C 180,E1 -4500.758,E2 -4500.758} C_VEL
LIN {X 0,Y 531.103,Z 482.956,A -85,B 0,C 180,E1 -4503.034,E2 -4503.034} C_VEL
LIN {X 0,Y 531.084,Z 482.959,A -85,B 0,C 180,E1 -4506.077,E2 -4506.077} C_VEL
LIN {X 0,Y 531.028,Z 482.965,A -85,B 0,C 180,E1 -4509.139,E2 -4509.139} C_VEL
LIN {X 0,Y 531.032,Z 482.964,A -85,B 0,C 180,E1 -4512.225,E2 -4512.225} C_VEL
LIN {X 0,Y 530.988,Z 482.97,A -85,B 0,C 180,E1 -4515.35,E2 -4515.35} C_VEL
LIN {X 0,Y 531.008,Z 482.967,A -85,B 0,C 180,E1 -4517.723,E2 -4517.723} C_VEL
LIN {X 0,Y 530.994,Z 482.968,A -85,B 0,C 180,E1 -4520.939,E2 -4520.939} C_VEL
LIN {X 0,Y 530.972,Z 482.971,A -85,B 0,C 180,E1 -4524.225,E2 -4524.225} C_VEL
LIN {X 0,Y 531.006,Z 482.967,A -85,B 0,C 180,E1 -4526.744,E2 -4526.744} C_VEL
LIN {X 0,Y 530.994,Z 482.971,A -85,B 0,C 180,E1 -4529.322,E2 -4529.322} C_VEL
LIN {X 0,Y 530.974,Z 482.971,A -85,B 0,C 180,E1 -4532.104,E2 -4532.104} C_VEL
LIN {X 0,Y 530.986,Z 482.971,A -85,B 0,C 180,E1 -4534.856,E2 -4534.856} C_VEL
LIN {X 0,Y 530.962,Z 482.973,A -85,B 0,C 180,E1 -4537.509,E2 -4537.509} C_VEL
LIN {X 0,Y 531.024,Z 482.965,A -85,B 0,C 180,E1 -4540.43,E2 -4540.43} C_VEL
LIN {X 0,Y 530.963,Z 482.975,A -85,B 0,C 180,E1 -4543.495,E2 -4543.495} C_VEL
LIN {X 0,Y 530.959,Z 482.974,A -85,B 0,C 180,E1 -4543.579,E2 -4543.579} C_VEL
LIN {X 0,Y 530.287,Z 483.057,A -85,B 0,C 180,E1 -4544.212,E2 -4544.212} C_VEL
LIN {X 0,Y 527.44,Z 483.411,A -85,B 0,C 180,E1 -4545.241,E2 -4545.241} C_VEL
LIN {X 0,Y 525.037,Z 483.712,A -85,B 0,C 180,E1 -4546.07,E2 -4546.07} C_VEL
LIN {X 0,Y 524.004,Z 483.84,A -85,B 0,C 180,E1 -4546.709,E2 -4546.709} C_VEL
LIN {X 0,Y 523.92,Z 483.85,A -85,B 0,C 180,E1 -4546.926,E2 -4546.926} C_VEL
LIN {X 0,Y 523.977,Z 483.844,A -85,B 0,C 180,E1 -4549.925,E2 -4549.925} C_VEL
LIN {X 0,Y 523.911,Z 483.85,A -85,B 0,C 180,E1 -4552.869,E2 -4552.869} C_VEL
LIN {X 0,Y 523.941,Z 483.849,A -85,B 0,C 180,E1 -4555.712,E2 -4555.712} C_VEL
LIN {X 0,Y 523.929,Z 483.848,A -85,B 0,C 180,E1 -4558.458,E2 -4558.458} C_VEL
LIN {X 0,Y 523.942,Z 483.848,A -85,B 0,C 180,E1 -4561.127,E2 -4561.127} C_VEL
LIN {X 0,Y 523.988,Z 483.842,A -85,B 0,C 180,E1 -4563.981,E2 -4563.981} C_VEL
LIN {X 0,Y 523.939,Z 483.848,A -85,B 0,C 180,E1 -4566.272,E2 -4566.272} C_VEL
LIN {X 0,Y 523.948,Z 483.846,A -85,B 0,C 180,E1 -4568.768,E2 -4568.768} C_VEL
LIN {X 0,Y 523.955,Z 483.847,A -85,B 0,C 180,E1 -4571.222,E2 -4571.222} C_VEL
LIN {X 0,Y 523.942,Z 483.848,A -85,B 0,C 180,E1 -4573.64,E2 -4573.64} C_VEL
LIN {X 0,Y 523.944,Z 483.847,A -85,B 0,C 180,E1 -4576.029,E2 -4576.029} C_VEL
LIN {X 0,Y 524.017,Z 483.838,A -85,B 0,C 180,E1 -4578.395,E2 -4578.395} C_VEL
LIN {X 0,Y 523.993,Z 483.841,A -85,B 0,C 180,E1 -4581.516,E2 -4581.516} C_VEL
LIN {X 0,Y 524.051,Z 483.834,A -85,B 0,C 180,E1 -4583.842,E2 -4583.842} C_VEL
LIN {X 0,Y 524.077,Z 483.83,A -85,B 0,C 180,E1 -4586.926,E2 -4586.926} C_VEL
LIN {X 0,Y 524.121,Z 483.825,A -85,B 0,C 180,E1 -4590,E2 -4590} C_VEL
LIN {X 0,Y 524.04,Z 483.836,A -85,B 0,C 180,E1 -4592.306,E2 -4592.306} C_VEL
LIN {X 0,Y 523.786,Z 483.87,A -85,B 0,C 180,E1 -4594.618,E2 -4594.618} C_VEL
LIN {X 0,Y 523.619,Z 486.549,A -85,B 0,C 180,E1 -4597.714,E2 -4597.714} C_VEL
LIN {X 0,Y 523.56,Z 489.467,A -85,B 0,C 180,E1 -4600.832,E2 -4600.832} C_VEL
LIN {X 0,Y 523.492,Z 492.408,A -85,B 0,C 180,E1 -4603.984,E2 -4603.984} C_VEL
LIN {X 0,Y 523.429,Z 494.651,A -85,B 0,C 180,E1 -4606.378,E2 -4606.378} C_VEL
LIN {X 0,Y 523.384,Z 496.951,A -85,B 0,C 180,E1 -4608.8,E2 -4608.8} C_VEL
LIN {X 0,Y 523.382,Z 498.929,A -85,B 0,C 180,E1 -4610.742,E2 -4610.742} C_VEL
LIN {X 0,Y 527.24,Z 513.95,A -85,B 0,C 180,E1 -4611.197,E2 -4611.197} C_VEL
LIN {X 0,Y 527.117,Z 527.726,A -85,B 0,C 180,E1 -4611.612,E2 -4611.612} C_VEL
LIN {X 0,Y 526.698,Z 542.231,A -85,B 0,C 180,E1 -4612.197,E2 -4612.197} C_VEL
LIN {X 0,Y 526.252,Z 556.385,A -85,B 0,C 180,E1 -4612.931,E2 -4612.931} C_VEL
LIN {X 0,Y 525.781,Z 569.081,A -85,B 0,C 180,E1 -4613.745,E2 -4613.745} C_VEL
LIN {X 0,Y 525.337,Z 581.306,A -85,B 0,C 180,E1 -4614.691,E2 -4614.691} C_VEL
LIN {X 0,Y 524.844,Z 593.272,A -85,B 0,C 180,E1 -4615.798,E2 -4615.798} C_VEL
LIN {X 0,Y 524.481,Z 603.222,A -85,B 0,C 180,E1 -4616.888,E2 -4616.888} C_VEL
LIN {X 0,Y 524.134,Z 613.395,A -85,B 0,C 180,E1 -4618.207,E2 -4618.207} C_VEL
LIN {X 0,Y 523.859,Z 621.805,A -85,B 0,C 180,E1 -4619.504,E2 -4619.504} C_VEL
LIN {X 0,Y 523.657,Z 628.867,A -85,B 0,C 180,E1 -4620.801,E2 -4620.801} C_VEL
LIN {X 0,Y 523.51,Z 635.351,A -85,B 0,C 180,E1 -4622.246,E2 -4622.246} C_VEL
LIN {X 0,Y 523.395,Z 641.419,A -85,B 0,C 180,E1 -4623.958,E2 -4623.958} C_VEL
LIN {X 0,Y 523.304,Z 644.944,A -85,B 0,C 180,E1 -4625.274,E2 -4625.274} C_VEL
LIN {X 0,Y 523.255,Z 647.09,A -85,B 0,C 180,E1 -4626.304,E2 -4626.304} C_VEL
LIN {X 0,Y 523.239,Z 649.027,A -85,B 0,C 180,E1 -4627.582,E2 -4627.582} C_VEL
LIN {X 0,Y 523.231,Z 650.303,A -85,B 0,C 180,E1 -4629.146,E2 -4629.146} C_VEL
LIN {X 0,Y 523.241,Z 650.486,A -85,B 0,C 180,E1 -4630.144,E2 -4630.144} C_VEL
LIN {X 0,Y 523.248,Z 650.135,A -85,B 0,C 180,E1 -4631.221,E2 -4631.221} C_VEL
LIN {X 0,Y 523.268,Z 649.165,A -85,B 0,C 180,E1 -4632.378,E2 -4632.378} C_VEL
LIN {X 0,Y 523.266,Z 647.613,A -85,B 0,C 180,E1 -4633.508,E2 -4633.508} C_VEL
LIN {X 0,Y 523.365,Z 645.386,A -85,B 0,C 180,E1 -4634.625,E2 -4634.625} C_VEL
LIN {X 0,Y 523.405,Z 641.461,A -85,B 0,C 180,E1 -4636.118,E2 -4636.118} C_VEL
LIN {X 0,Y 523.486,Z 636.369,A -85,B 0,C 180,E1 -4637.594,E2 -4637.594} C_VEL
LIN {X 0,Y 523.615,Z 629.653,A -85,B 0,C 180,E1 -4639.131,E2 -4639.131} C_VEL
LIN {X 0,Y 523.853,Z 621.38,A -85,B 0,C 180,E1 -4640.661,E2 -4640.661} C_VEL
LIN {X 0,Y 524.209,Z 611.684,A -85,B 0,C 180,E1 -4642.127,E2 -4642.127} C_VEL
LIN {X 0,Y 524.556,Z 600.683,A -85,B 0,C 180,E1 -4643.501,E2 -4643.501} C_VEL
LIN {X 0,Y 525.055,Z 588.753,A -85,B 0,C 180,E1 -4644.735,E2 -4644.735} C_VEL
LIN {X 0,Y 525.508,Z 576.071,A -85,B 0,C 180,E1 -4645.826,E2 -4645.826} C_VEL
LIN {X 0,Y 525.993,Z 562.58,A -85,B 0,C 180,E1 -4646.782,E2 -4646.782} C_VEL
LIN {X 0,Y 526.486,Z 548.851,A -85,B 0,C 180,E1 -4647.571,E2 -4647.571} C_VEL
LIN {X 0,Y 526.958,Z 534.835,A -85,B 0,C 180,E1 -4648.21,E2 -4648.21} C_VEL
LIN {X 0,Y 527.248,Z 520.247,A -85,B 0,C 180,E1 -4648.719,E2 -4648.719} C_VEL
LIN {X 0,Y 527.21,Z 513.838,A -85,B 0,C 180,E1 -4648.898,E2 -4648.898} C_VEL
LIN {X 0,Y 523.372,Z 498.75,A -85,B 0,C 180,E1 -4649.373,E2 -4649.373} C_VEL
LIN {X 0,Y 523.4,Z 495.957,A -85,B 0,C 180,E1 -4652.401,E2 -4652.401} C_VEL
LIN {X 0,Y 523.464,Z 493.33,A -85,B 0,C 180,E1 -4655.404,E2 -4655.404} C_VEL
LIN {X 0,Y 523.525,Z 491.265,A -85,B 0,C 180,E1 -4657.921,E2 -4657.921} C_VEL
LIN {X 0,Y 523.611,Z 489.077,A -85,B 0,C 180,E1 -4660.393,E2 -4660.393} C_VEL
LIN {X 0,Y 523.678,Z 486.945,A -85,B 0,C 180,E1 -4662.827,E2 -4662.827} C_VEL
LIN {X 0,Y 523.74,Z 484.812,A -85,B 0,C 180,E1 -4665.228,E2 -4665.228} C_VEL
LIN {X 0,Y 523.703,Z 484.103,A -85,B 0,C 180,E1 -4666.021,E2 -4666.021} C_VEL
LIN {X 0,Y 523.966,Z 483.847,A -85,B 0,C 180,E1 -4668.393,E2 -4668.393} C_VEL
LIN {X 0,Y 524.005,Z 483.837,A -85,B 0,C 180,E1 -4671.516,E2 -4671.516} C_VEL
LIN {X 0,Y 524.085,Z 483.825,A -85,B 0,C 180,E1 -4674.613,E2 -4674.613} C_VEL
LIN {X 0,Y 524.109,Z 483.829,A -85,B 0,C 180,E1 -4677.694,E2 -4677.694} C_VEL
LIN {X 0,Y 524.12,Z 483.82,A -85,B 0,C 180,E1 -4680.768,E2 -4680.768} C_VEL
LIN {X 0,Y 524.07,Z 483.83,A -85,B 0,C 180,E1 -4683.075,E2 -4683.075} C_VEL
LIN {X 0,Y 524.043,Z 483.83,A -85,B 0,C 180,E1 -4686.159,E2 -4686.159} C_VEL
LIN {X 0,Y 523.997,Z 483.841,A -85,B 0,C 180,E1 -4689.262,E2 -4689.262} C_VEL
LIN {X 0,Y 524.004,Z 483.834,A -85,B 0,C 180,E1 -4691.743,E2 -4691.743} C_VEL
LIN {X 0,Y 523.988,Z 483.841,A -85,B 0,C 180,E1 -4695.052,E2 -4695.052} C_VEL
LIN {X 0,Y 523.96,Z 483.84,A -85,B 0,C 180,E1 -4697.969,E2 -4697.969} C_VEL
LIN {X 0,Y 523.968,Z 483.845,A -85,B 0,C 180,E1 -4700.41,E2 -4700.41} C_VEL
LIN {X 0,Y 523.913,Z 483.847,A -85,B 0,C 180,E1 -4702.893,E2 -4702.893} C_VEL
LIN {X 0,Y 523.951,Z 483.841,A -85,B 0,C 180,E1 -4705.419,E2 -4705.419} C_VEL
LIN {X 0,Y 523.967,Z 483.846,A -85,B 0,C 180,E1 -4707.999,E2 -4707.999} C_VEL
LIN {X 0,Y 523.949,Z 483.842,A -85,B 0,C 180,E1 -4710.856,E2 -4710.856} C_VEL
LIN {X 0,Y 523.958,Z 483.847,A -85,B 0,C 180,E1 -4713.735,E2 -4713.735} C_VEL
LIN {X 0,Y 523.92,Z 483.847,A -85,B 0,C 180,E1 -4716.404,E2 -4716.404} C_VEL
LIN {X 0,Y 523.921,Z 483.846,A -85,B 0,C 180,E1 -4719.085,E2 -4719.085} C_VEL
LIN {X 0,Y 523.955,Z 483.844,A -85,B 0,C 180,E1 -4722.118,E2 -4722.118} C_VEL
LIN {X 0,Y 523.954,Z 483.868,A -85,B 0,C 180,E1 -4725.137,E2 -4725.137} C_VEL
LIN {X 0,Y 524.962,Z 489.816,A -85,B 0,C 180,E1 -4727.981,E2 -4727.981} C_VEL
LIN {X 0,Y 525.013,Z 494.565,A -85,B 0,C 180,E1 -4730.019,E2 -4730.019} C_VEL
LIN {X 0,Y 524.735,Z 501.87,A -85,B 0,C 180,E1 -4732.936,E2 -4732.936} C_VEL
LIN {X 0,Y 524.609,Z 508.098,A -85,B 0,C 180,E1 -4735.295,E2 -4735.295} C_VEL
LIN {X 0,Y 524.453,Z 516.995,A -85,B 0,C 180,E1 -4738.492,E2 -4738.492} C_VEL
LIN {X 0,Y 524.244,Z 525.98,A -85,B 0,C 180,E1 -4741.581,E2 -4741.581} C_VEL
LIN {X 0,Y 524.108,Z 534.032,A -85,B 0,C 180,E1 -4744.267,E2 -4744.267} C_VEL
LIN {X 0,Y 523.983,Z 543.003,A -85,B 0,C 180,E1 -4747.11,E2 -4747.11} C_VEL
LIN {X 0,Y 523.882,Z 551.893,A -85,B 0,C 180,E1 -4749.895,E2 -4749.895} C_VEL
LIN {X 0,Y 523.877,Z 554.326,A -85,B 0,C 180,E1 -4750.653,E2 -4750.653} C_VEL
LIN {X 0,Y 527.485,Z 569.476,A -85,B 0,C 180,E1 -4751.059,E2 -4751.059} C_VEL
LIN {X 0,Y 527.168,Z 584.768,A -85,B 0,C 180,E1 -4751.474,E2 -4751.474} C_VEL
LIN {X 0,Y 526.78,Z 599.985,A -85,B 0,C 180,E1 -4752.055,E2 -4752.055} C_VEL
LIN {X 0,Y 526.392,Z 613.359,A -85,B 0,C 180,E1 -4752.718,E2 -4752.718} C_VEL
LIN {X 0,Y 525.926,Z 626.192,A -85,B 0,C 180,E1 -4753.503,E2 -4753.503} C_VEL
LIN {X 0,Y 525.422,Z 639.346,A -85,B 0,C 180,E1 -4754.483,E2 -4754.483} C_VEL
LIN {X 0,Y 524.98,Z 650.374,A -85,B 0,C 180,E1 -4755.463,E2 -4755.463} C_VEL
LIN {X 0,Y 524.598,Z 661.507,A -85,B 0,C 180,E1 -4756.638,E2 -4756.638} C_VEL
LIN {X 0,Y 524.154,Z 672.308,A -85,B 0,C 180,E1 -4758.005,E2 -4758.005} C_VEL
LIN {X 0,Y 523.943,Z 681.295,A -85,B 0,C 180,E1 -4759.371,E2 -4759.371} C_VEL
LIN {X 0,Y 523.699,Z 688.748,A -85,B 0,C 180,E1 -4760.733,E2 -4760.733} C_VEL
LIN {X 0,Y 523.535,Z 695.699,A -85,B 0,C 180,E1 -4762.285,E2 -4762.285} C_VEL
LIN {X 0,Y 523.436,Z 701.162,A -85,B 0,C 180,E1 -4763.834,E2 -4763.834} C_VEL
LIN {X 0,Y 523.323,Z 705.29,A -85,B 0,C 180,E1 -4765.378,E2 -4765.378} C_VEL
LIN {X 0,Y 523.358,Z 708.184,A -85,B 0,C 180,E1 -4766.921,E2 -4766.921} C_VEL
LIN {X 0,Y 523.272,Z 709.909,A -85,B 0,C 180,E1 -4768.46,E2 -4768.46} C_VEL
LIN {X 0,Y 523.243,Z 710.5,A -85,B 0,C 180,E1 -4770,E2 -4770} C_VEL
LIN {X 0,Y 523.272,Z 709.908,A -85,B 0,C 180,E1 -4771.539,E2 -4771.539} C_VEL
LIN {X 0,Y 523.358,Z 708.181,A -85,B 0,C 180,E1 -4773.079,E2 -4773.079} C_VEL
LIN {X 0,Y 523.323,Z 705.29,A -85,B 0,C 180,E1 -4774.621,E2 -4774.621} C_VEL
LIN {X 0,Y 523.43,Z 701.167,A -85,B 0,C 180,E1 -4776.166,E2 -4776.166} C_VEL
LIN {X 0,Y 523.534,Z 695.703,A -85,B 0,C 180,E1 -4777.714,E2 -4777.714} C_VEL
LIN {X 0,Y 523.699,Z 688.747,A -85,B 0,C 180,E1 -4779.267,E2 -4779.267} C_VEL
LIN {X 0,Y 523.986,Z 680.086,A -85,B 0,C 180,E1 -4780.822,E2 -4780.822} C_VEL
LIN {X 0,Y 524.231,Z 670.851,A -85,B 0,C 180,E1 -4782.193,E2 -4782.193} C_VEL
LIN {X 0,Y 524.597,Z 661.513,A -85,B 0,C 180,E1 -4783.361,E2 -4783.361} C_VEL
LIN {X 0,Y 525.036,Z 649.367,A -85,B 0,C 180,E1 -4784.634,E2 -4784.634} C_VEL
LIN {X 0,Y 525.481,Z 637.834,A -85,B 0,C 180,E1 -4785.644,E2 -4785.644} C_VEL
LIN {X 0,Y 525.929,Z 624.777,A -85,B 0,C 180,E1 -4786.596,E2 -4786.596} C_VEL
LIN {X 0,Y 526.446,Z 611.6,A -85,B 0,C 180,E1 -4787.379,E2 -4787.379} C_VEL
LIN {X 0,Y 526.835,Z 598.31,A -85,B 0,C 180,E1 -4788.018,E2 -4788.018} C_VEL
LIN {X 0,Y 527.201,Z 583.52,A -85,B 0,C 180,E1 -4788.567,E2 -4788.567} C_VEL
LIN {X 0,Y 527.405,Z 569.189,A -85,B 0,C 180,E1 -4788.95,E2 -4788.95} C_VEL
LIN {X 0,Y 523.874,Z 554.352,A -85,B 0,C 180,E1 -4789.346,E2 -4789.346} C_VEL
LIN {X 0,Y 523.978,Z 545.206,A -85,B 0,C 180,E1 -4792.259,E2 -4792.259} C_VEL
LIN {X 0,Y 524.137,Z 535.458,A -85,B 0,C 180,E1 -4795.408,E2 -4795.408} C_VEL
LIN {X 0,Y 524.298,Z 526.439,A -85,B 0,C 180,E1 -4798.415,E2 -4798.415} C_VEL
LIN {X 0,Y 524.501,Z 517.648,A -85,B 0,C 180,E1 -4801.504,E2 -4801.504} C_VEL
LIN {X 0,Y 524.652,Z 510.089,A -85,B 0,C 180,E1 -4804.235,E2 -4804.235} C_VEL
LIN {X 0,Y 524.857,Z 502.628,A -85,B 0,C 180,E1 -4807.052,E2 -4807.052} C_VEL
LIN {X 0,Y 525.137,Z 495.231,A -85,B 0,C 180,E1 -4809.969,E2 -4809.969} C_VEL
LIN {X 0,Y 525.087,Z 490.349,A -85,B 0,C 180,E1 -4812.006,E2 -4812.006} C_VEL
LIN {X 0,Y 524.048,Z 484.395,A -85,B 0,C 180,E1 -4814.702,E2 -4814.702} C_VEL
LIN {X 0,Y 523.948,Z 483.845,A -85,B 0,C 180,E1 -4815.033,E2 -4815.033} C_VEL
LIN {X 0,Y 523.958,Z 483.846,A -85,B 0,C 180,E1 -4817.882,E2 -4817.882} C_VEL
LIN {X 0,Y 523.953,Z 483.848,A -85,B 0,C 180,E1 -4820.918,E2 -4820.918} C_VEL
LIN {X 0,Y 523.92,Z 483.85,A -85,B 0,C 180,E1 -4823.827,E2 -4823.827} C_VEL
LIN {X 0,Y 523.935,Z 483.849,A -85,B 0,C 180,E1 -4826.635,E2 -4826.635} C_VEL
LIN {X 0,Y 523.954,Z 483.846,A -85,B 0,C 180,E1 -4829.356,E2 -4829.356} C_VEL
LIN {X 0,Y 523.971,Z 483.842,A -85,B 0,C 180,E1 -4832.28,E2 -4832.28} C_VEL
LIN {X 0,Y 523.945,Z 483.846,A -85,B 0,C 180,E1 -4834.581,E2 -4834.581} C_VEL
LIN {X 0,Y 523.907,Z 483.851,A -85,B 0,C 180,E1 -4837.106,E2 -4837.106} C_VEL
LIN {X 0,Y 523.969,Z 483.844,A -85,B 0,C 180,E1 -4839.865,E2 -4839.865} C_VEL
LIN {X 0,Y 523.961,Z 483.845,A -85,B 0,C 180,E1 -4842.837,E2 -4842.837} C_VEL
LIN {X 0,Y 523.965,Z 483.847,A -85,B 0,C 180,E1 -4845.236,E2 -4845.236} C_VEL
LIN {X 0,Y 524.001,Z 483.84,A -85,B 0,C 180,E1 -4848.394,E2 -4848.394} C_VEL
LIN {X 0,Y 524,Z 483.841,A -85,B 0,C 180,E1 -4851.516,E2 -4851.516} C_VEL
LIN {X 0,Y 524.091,Z 483.827,A -85,B 0,C 180,E1 -4854.614,E2 -4854.614} C_VEL
LIN {X 0,Y 524.104,Z 483.827,A -85,B 0,C 180,E1 -4857.695,E2 -4857.695} C_VEL
LIN {X 0,Y 524.116,Z 483.826,A -85,B 0,C 180,E1 -4860.769,E2 -4860.769} C_VEL
LIN {X 0,Y 524.07,Z 483.832,A -85,B 0,C 180,E1 -4863.075,E2 -4863.075} C_VEL
LIN {X 0,Y 524.044,Z 483.835,A -85,B 0,C 180,E1 -4866.159,E2 -4866.159} C_VEL
